PROGRAM AxisHorzMovementOutputCtrl_Arm1
VAR

	LdUnhook: CMP_OC_DW;
	Stn1Unhook: CMP_OC_DW;
	Stn2Unhook: CMP_OC_DW;
	Stn3Unhook: CMP_OC_DW;
	Stn4Unhook: CMP_OC_DW;
	Stn5Unhook: CMP_OC_DW;
	Stn6Unhook: CMP_OC_DW;
	Stn7Unhook: CMP_OC_DW;
	Stn8Unhook: CMP_OC_DW;
	Stn9Unhook: CMP_OC_DW;
	Stn10Unhook: CMP_OC_DW;
	Stn11Unhook: CMP_OC_DW;
	Stn12Unhook: CMP_OC_DW;
	Uld1Unhook: CMP_OC_DW;
	Uld2Unhook: CMP_OC_DW;

	LdHook: CMP_OC_DW;
	Stn1Hook: CMP_OC_DW;
	Stn2Hook: CMP_OC_DW;
	Stn3Hook: CMP_OC_DW;
	Stn4Hook: CMP_OC_DW;
	Stn5Hook: CMP_OC_DW;
	Stn6Hook: CMP_OC_DW;
	Stn7Hook: CMP_OC_DW;
	Stn8Hook: CMP_OC_DW;
	Stn9Hook: CMP_OC_DW;
	Stn10Hook: CMP_OC_DW;
	Stn11Hook: CMP_OC_DW;
	Stn12Hook: CMP_OC_DW;
	Uld1Hook: CMP_OC_DW;
	Uld2Hook: CMP_OC_DW;

END_VAR

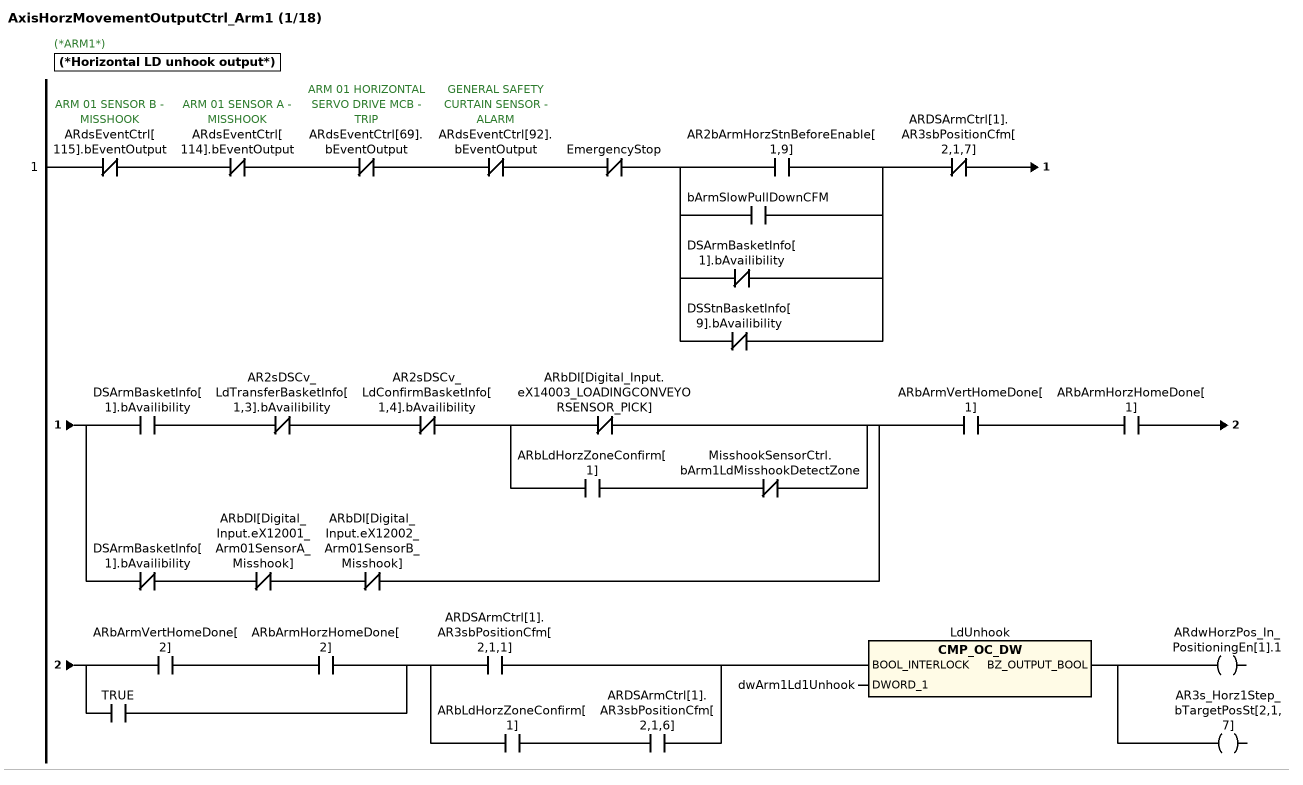
// NETWORK 1
// (*ARM1*)
//   ARdsEventCtrl[115].bEventOutput: ARM 01 SENSOR B - MISSHOOK
//   ARdsEventCtrl[114].bEventOutput: ARM 01 SENSOR A - MISSHOOK
//   ARdsEventCtrl[69].bEventOutput: ARM 01 HORIZONTAL SERVO DRIVE MCB - TRIP
//   ARdsEventCtrl[92].bEventOutput: GENERAL SAFETY CURTAIN SENSOR - ALARM
// label: (*Horizontal LD unhook output*)
LdUnhook(BOOL_INTERLOCK := (((NOT ARdsEventCtrl[115].bEventOutput AND NOT ARdsEventCtrl[114].bEventOutput AND NOT ARdsEventCtrl[69].bEventOutput AND NOT ARdsEventCtrl[92].bEventOutput AND NOT EmergencyStop) AND (AR2bArmHorzStnBeforeEnable[1,9] OR bArmSlowPullDownCFM OR NOT DSArmBasketInfo[1].bAvailibility OR NOT DSStnBasketInfo[9].bAvailibility)) AND NOT ARDSArmCtrl[1].AR3sbPositionCfm[2,1,7] AND (DSArmBasketInfo[1].bAvailibility AND NOT AR2sDSCv_LdTransferBasketInfo[1,3].bAvailibility AND NOT AR2sDSCv_LdConfirmBasketInfo[1,4].bAvailibility AND (NOT ARbDI[Digital_Input.eX14003_LOADINGCONVEYORSENSOR_PICK] OR ARbLdHorzZoneConfirm[1] AND NOT MisshookSensorCtrl.bArm1LdMisshookDetectZone) OR NOT DSArmBasketInfo[1].bAvailibility AND NOT ARbDI[Digital_Input.eX12001_Arm01SensorA_Misshook] AND NOT ARbDI[Digital_Input.eX12002_Arm01SensorB_Misshook])) AND ARbArmVertHomeDone[1] AND ARbArmHorzHomeDone[1] AND (ARbArmVertHomeDone[2] AND ARbArmHorzHomeDone[2] OR TRUE) AND (ARDSArmCtrl[1].AR3sbPositionCfm[2,1,1] OR ARbLdHorzZoneConfirm[1] AND ARDSArmCtrl[1].AR3sbPositionCfm[2,1,6]), DWORD_1 := dwArm1Ld1Unhook); // CMP_OC_DW
ARdwHorzPos_In_PositioningEn[1].1 := LdUnhook.BZ_OUTPUT_BOOL;
AR3s_Horz1Step_bTargetPosSt[2,1,7] := LdUnhook.BZ_OUTPUT_BOOL;

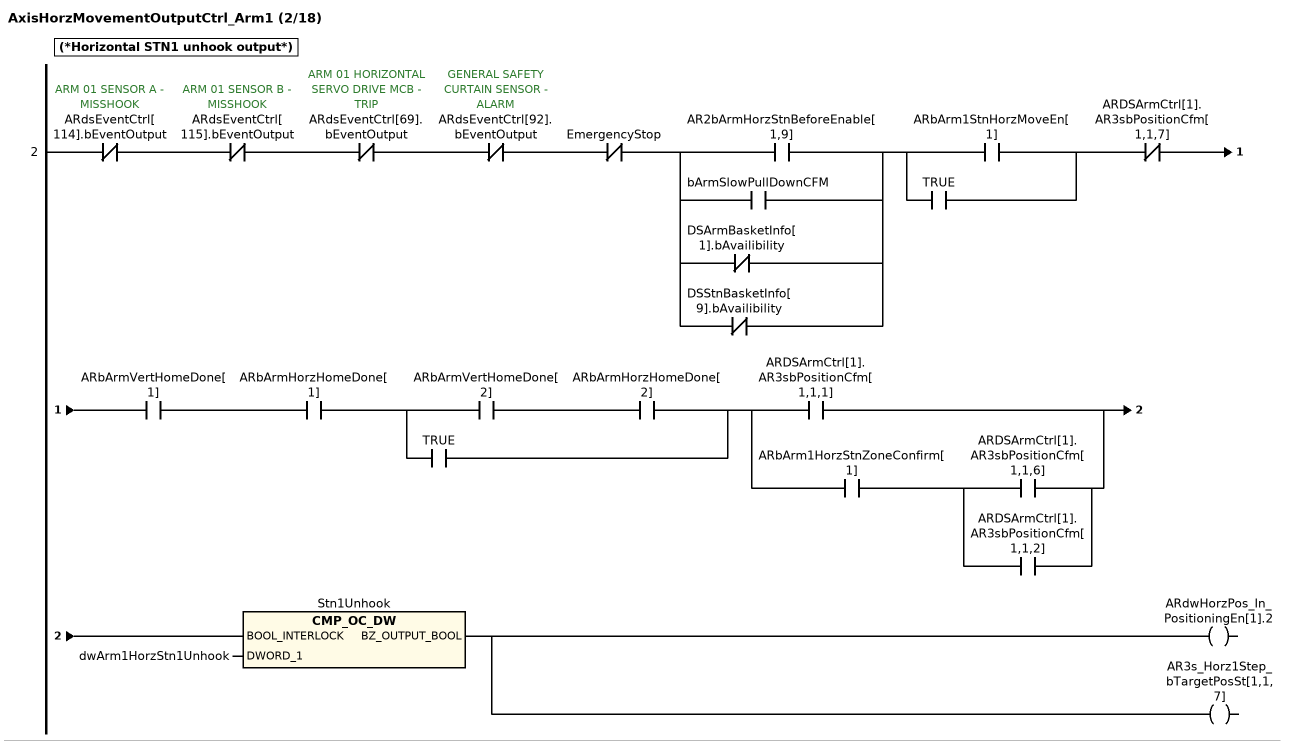
// NETWORK 2
//   ARdsEventCtrl[114].bEventOutput: ARM 01 SENSOR A - MISSHOOK
//   ARdsEventCtrl[115].bEventOutput: ARM 01 SENSOR B - MISSHOOK
//   ARdsEventCtrl[69].bEventOutput: ARM 01 HORIZONTAL SERVO DRIVE MCB - TRIP
//   ARdsEventCtrl[92].bEventOutput: GENERAL SAFETY CURTAIN SENSOR - ALARM
// label: (*Horizontal STN1 unhook output*)
Stn1Unhook(BOOL_INTERLOCK := ((NOT ARdsEventCtrl[114].bEventOutput AND NOT ARdsEventCtrl[115].bEventOutput AND NOT ARdsEventCtrl[69].bEventOutput AND NOT ARdsEventCtrl[92].bEventOutput AND NOT EmergencyStop) AND (AR2bArmHorzStnBeforeEnable[1,9] OR bArmSlowPullDownCFM OR NOT DSArmBasketInfo[1].bAvailibility OR NOT DSStnBasketInfo[9].bAvailibility) AND (ARbArm1StnHorzMoveEn[1] OR TRUE)) AND NOT ARDSArmCtrl[1].AR3sbPositionCfm[1,1,7] AND ARbArmVertHomeDone[1] AND ARbArmHorzHomeDone[1] AND (ARbArmVertHomeDone[2] AND ARbArmHorzHomeDone[2] OR TRUE) AND (ARDSArmCtrl[1].AR3sbPositionCfm[1,1,1] OR ARbArm1HorzStnZoneConfirm[1] AND (ARDSArmCtrl[1].AR3sbPositionCfm[1,1,6] OR ARDSArmCtrl[1].AR3sbPositionCfm[1,1,2])), DWORD_1 := dwArm1HorzStn1Unhook); // CMP_OC_DW
ARdwHorzPos_In_PositioningEn[1].2 := Stn1Unhook.BZ_OUTPUT_BOOL;
AR3s_Horz1Step_bTargetPosSt[1,1,7] := Stn1Unhook.BZ_OUTPUT_BOOL;

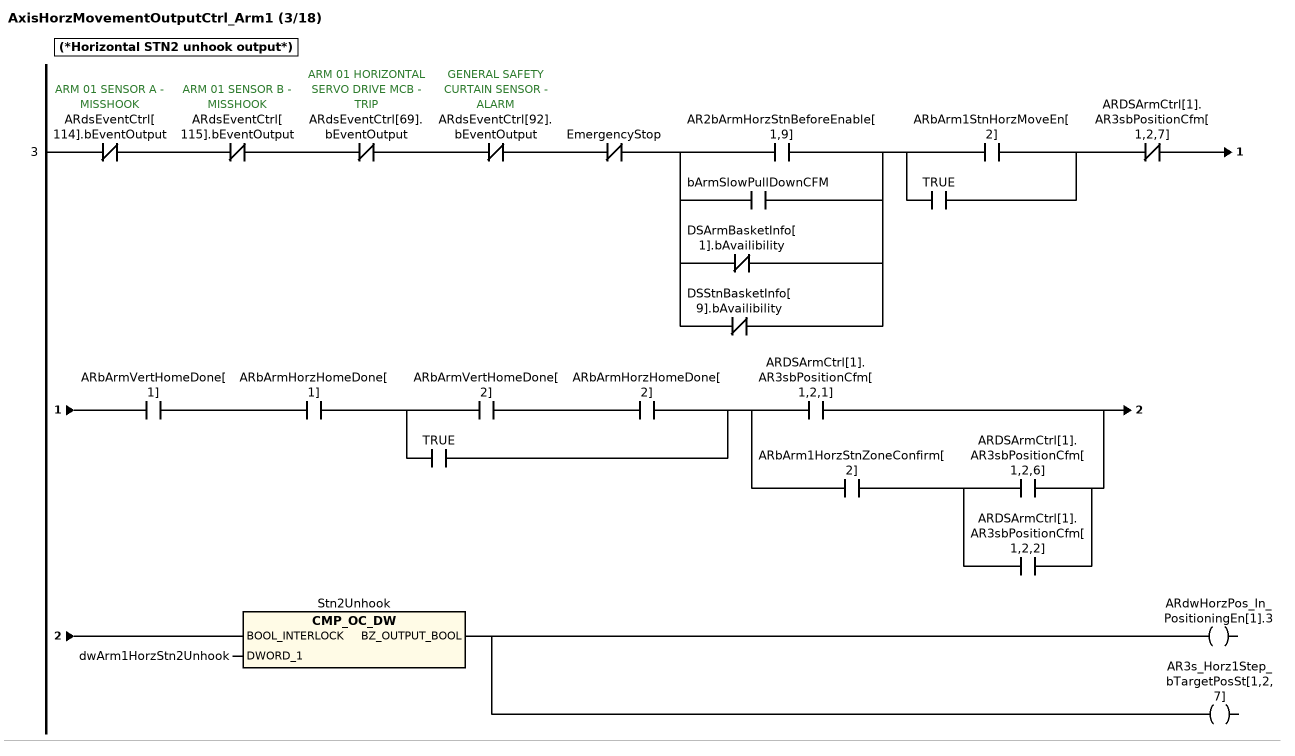
// NETWORK 3
//   ARdsEventCtrl[114].bEventOutput: ARM 01 SENSOR A - MISSHOOK
//   ARdsEventCtrl[115].bEventOutput: ARM 01 SENSOR B - MISSHOOK
//   ARdsEventCtrl[69].bEventOutput: ARM 01 HORIZONTAL SERVO DRIVE MCB - TRIP
//   ARdsEventCtrl[92].bEventOutput: GENERAL SAFETY CURTAIN SENSOR - ALARM
// label: (*Horizontal STN2 unhook output*)
Stn2Unhook(BOOL_INTERLOCK := ((NOT ARdsEventCtrl[114].bEventOutput AND NOT ARdsEventCtrl[115].bEventOutput AND NOT ARdsEventCtrl[69].bEventOutput AND NOT ARdsEventCtrl[92].bEventOutput AND NOT EmergencyStop) AND (AR2bArmHorzStnBeforeEnable[1,9] OR bArmSlowPullDownCFM OR NOT DSArmBasketInfo[1].bAvailibility OR NOT DSStnBasketInfo[9].bAvailibility) AND (ARbArm1StnHorzMoveEn[2] OR TRUE)) AND NOT ARDSArmCtrl[1].AR3sbPositionCfm[1,2,7] AND ARbArmVertHomeDone[1] AND ARbArmHorzHomeDone[1] AND (ARbArmVertHomeDone[2] AND ARbArmHorzHomeDone[2] OR TRUE) AND (ARDSArmCtrl[1].AR3sbPositionCfm[1,2,1] OR ARbArm1HorzStnZoneConfirm[2] AND (ARDSArmCtrl[1].AR3sbPositionCfm[1,2,6] OR ARDSArmCtrl[1].AR3sbPositionCfm[1,2,2])), DWORD_1 := dwArm1HorzStn2Unhook); // CMP_OC_DW
ARdwHorzPos_In_PositioningEn[1].3 := Stn2Unhook.BZ_OUTPUT_BOOL;
AR3s_Horz1Step_bTargetPosSt[1,2,7] := Stn2Unhook.BZ_OUTPUT_BOOL;

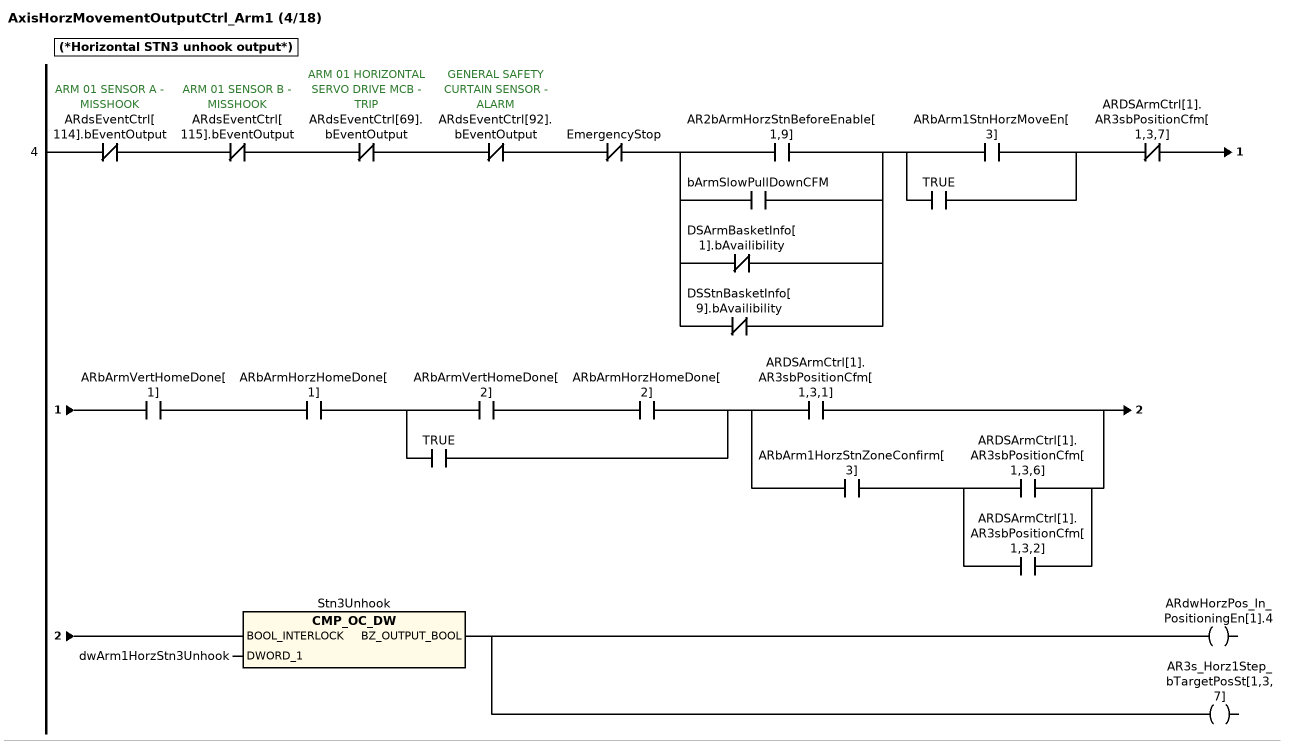
// NETWORK 4
//   ARdsEventCtrl[114].bEventOutput: ARM 01 SENSOR A - MISSHOOK
//   ARdsEventCtrl[115].bEventOutput: ARM 01 SENSOR B - MISSHOOK
//   ARdsEventCtrl[69].bEventOutput: ARM 01 HORIZONTAL SERVO DRIVE MCB - TRIP
//   ARdsEventCtrl[92].bEventOutput: GENERAL SAFETY CURTAIN SENSOR - ALARM
// label: (*Horizontal STN3 unhook output*)
Stn3Unhook(BOOL_INTERLOCK := ((NOT ARdsEventCtrl[114].bEventOutput AND NOT ARdsEventCtrl[115].bEventOutput AND NOT ARdsEventCtrl[69].bEventOutput AND NOT ARdsEventCtrl[92].bEventOutput AND NOT EmergencyStop) AND (AR2bArmHorzStnBeforeEnable[1,9] OR bArmSlowPullDownCFM OR NOT DSArmBasketInfo[1].bAvailibility OR NOT DSStnBasketInfo[9].bAvailibility) AND (ARbArm1StnHorzMoveEn[3] OR TRUE)) AND NOT ARDSArmCtrl[1].AR3sbPositionCfm[1,3,7] AND ARbArmVertHomeDone[1] AND ARbArmHorzHomeDone[1] AND (ARbArmVertHomeDone[2] AND ARbArmHorzHomeDone[2] OR TRUE) AND (ARDSArmCtrl[1].AR3sbPositionCfm[1,3,1] OR ARbArm1HorzStnZoneConfirm[3] AND (ARDSArmCtrl[1].AR3sbPositionCfm[1,3,6] OR ARDSArmCtrl[1].AR3sbPositionCfm[1,3,2])), DWORD_1 := dwArm1HorzStn3Unhook); // CMP_OC_DW
ARdwHorzPos_In_PositioningEn[1].4 := Stn3Unhook.BZ_OUTPUT_BOOL;
AR3s_Horz1Step_bTargetPosSt[1,3,7] := Stn3Unhook.BZ_OUTPUT_BOOL;

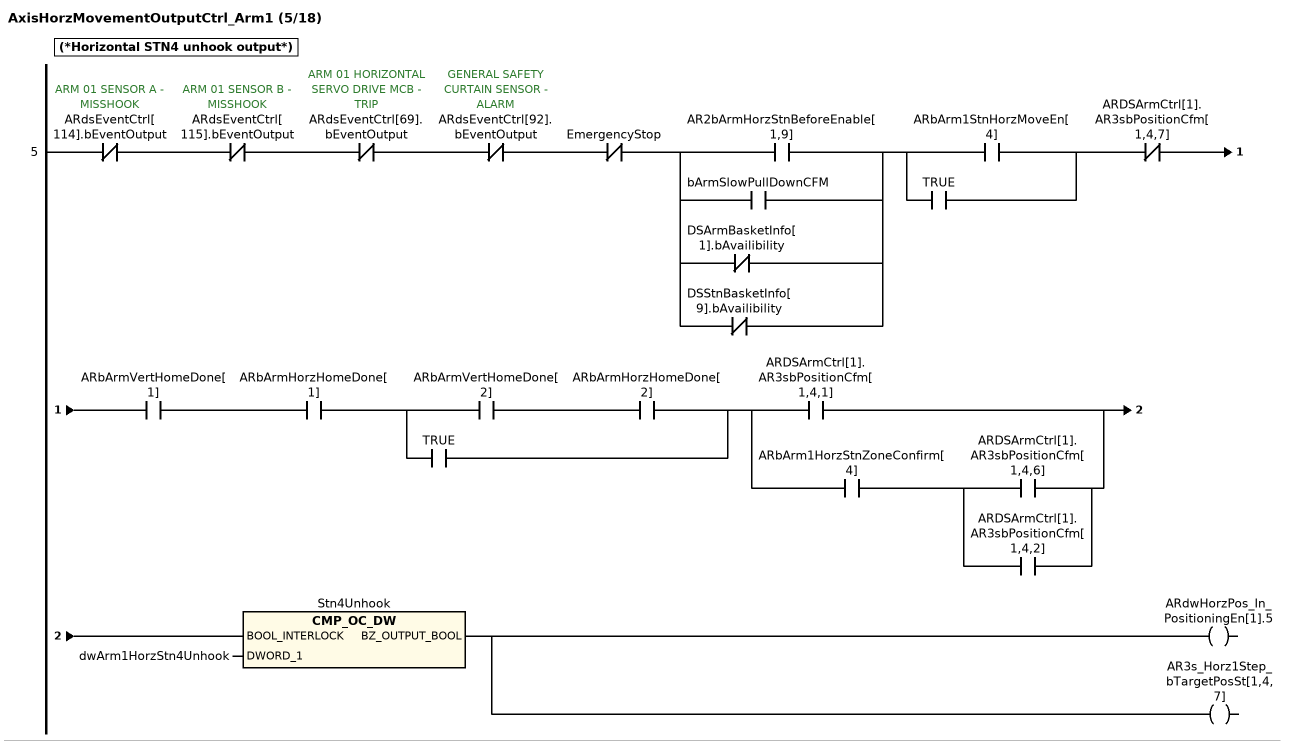
// NETWORK 5
//   ARdsEventCtrl[114].bEventOutput: ARM 01 SENSOR A - MISSHOOK
//   ARdsEventCtrl[115].bEventOutput: ARM 01 SENSOR B - MISSHOOK
//   ARdsEventCtrl[69].bEventOutput: ARM 01 HORIZONTAL SERVO DRIVE MCB - TRIP
//   ARdsEventCtrl[92].bEventOutput: GENERAL SAFETY CURTAIN SENSOR - ALARM
// label: (*Horizontal STN4 unhook output*)
Stn4Unhook(BOOL_INTERLOCK := ((NOT ARdsEventCtrl[114].bEventOutput AND NOT ARdsEventCtrl[115].bEventOutput AND NOT ARdsEventCtrl[69].bEventOutput AND NOT ARdsEventCtrl[92].bEventOutput AND NOT EmergencyStop) AND (AR2bArmHorzStnBeforeEnable[1,9] OR bArmSlowPullDownCFM OR NOT DSArmBasketInfo[1].bAvailibility OR NOT DSStnBasketInfo[9].bAvailibility) AND (ARbArm1StnHorzMoveEn[4] OR TRUE)) AND NOT ARDSArmCtrl[1].AR3sbPositionCfm[1,4,7] AND ARbArmVertHomeDone[1] AND ARbArmHorzHomeDone[1] AND (ARbArmVertHomeDone[2] AND ARbArmHorzHomeDone[2] OR TRUE) AND (ARDSArmCtrl[1].AR3sbPositionCfm[1,4,1] OR ARbArm1HorzStnZoneConfirm[4] AND (ARDSArmCtrl[1].AR3sbPositionCfm[1,4,6] OR ARDSArmCtrl[1].AR3sbPositionCfm[1,4,2])), DWORD_1 := dwArm1HorzStn4Unhook); // CMP_OC_DW
ARdwHorzPos_In_PositioningEn[1].5 := Stn4Unhook.BZ_OUTPUT_BOOL;
AR3s_Horz1Step_bTargetPosSt[1,4,7] := Stn4Unhook.BZ_OUTPUT_BOOL;

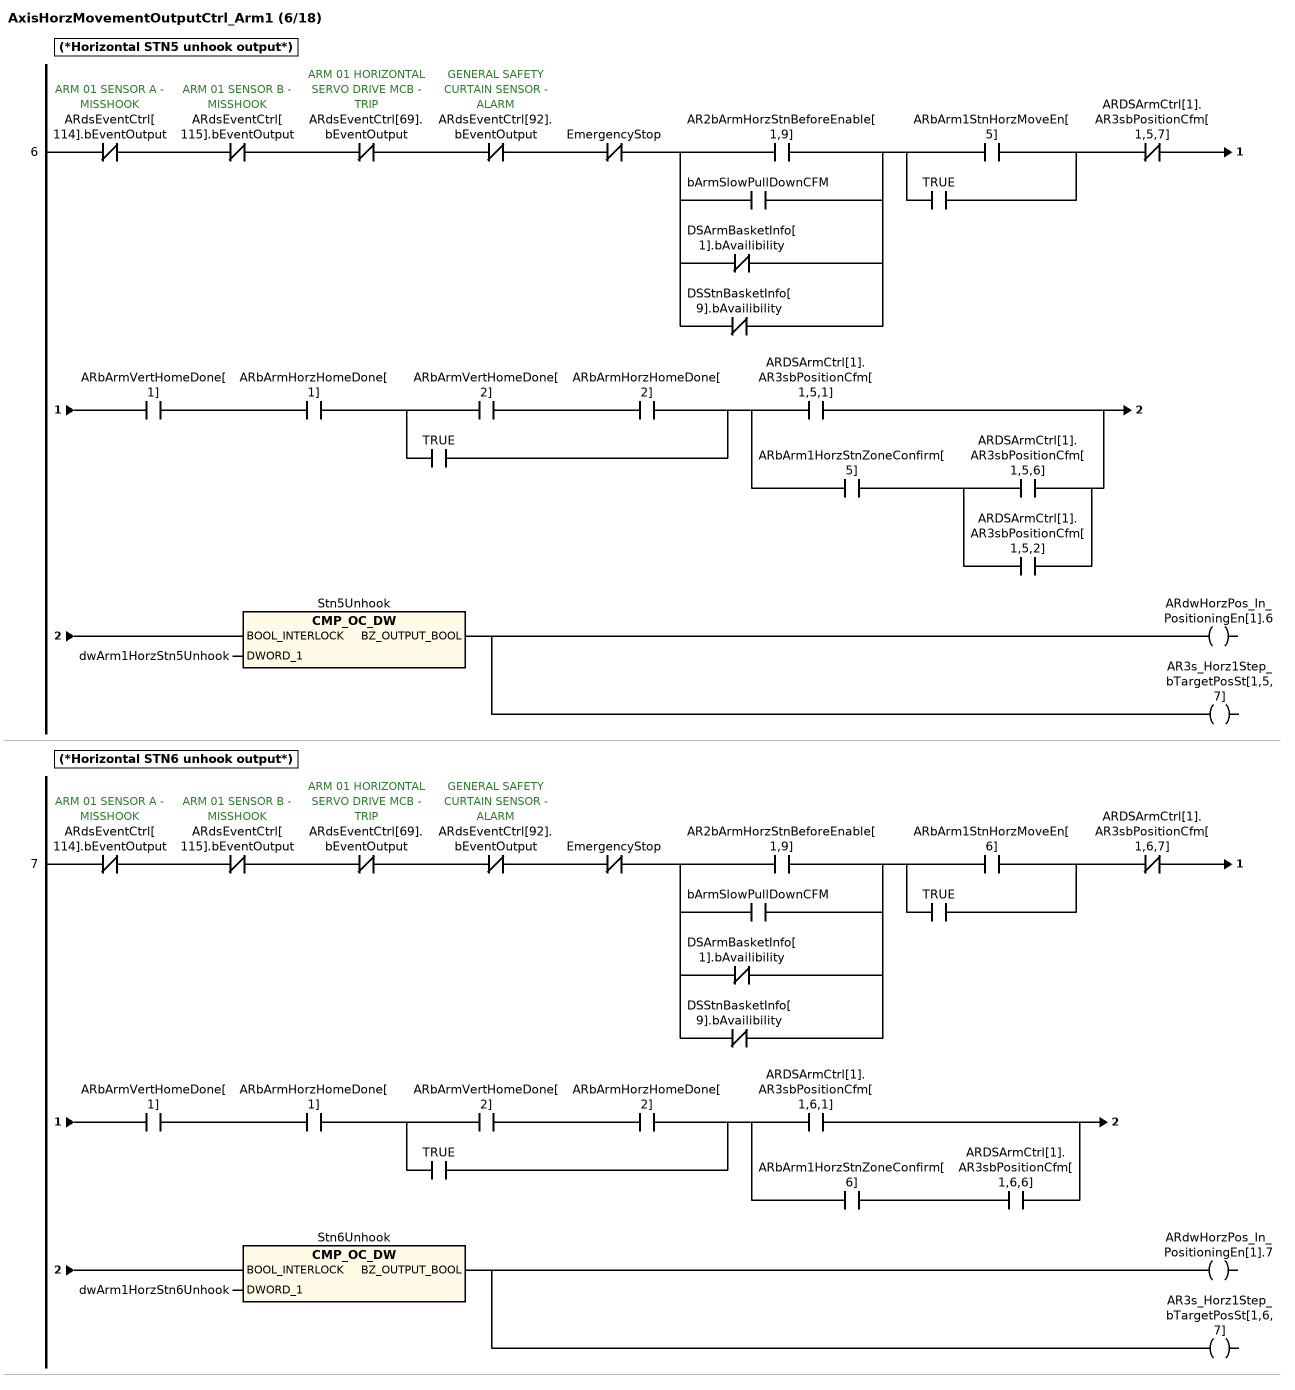
// NETWORK 6
//   ARdsEventCtrl[114].bEventOutput: ARM 01 SENSOR A - MISSHOOK
//   ARdsEventCtrl[115].bEventOutput: ARM 01 SENSOR B - MISSHOOK
//   ARdsEventCtrl[69].bEventOutput: ARM 01 HORIZONTAL SERVO DRIVE MCB - TRIP
//   ARdsEventCtrl[92].bEventOutput: GENERAL SAFETY CURTAIN SENSOR - ALARM
// label: (*Horizontal STN5 unhook output*)
Stn5Unhook(BOOL_INTERLOCK := ((NOT ARdsEventCtrl[114].bEventOutput AND NOT ARdsEventCtrl[115].bEventOutput AND NOT ARdsEventCtrl[69].bEventOutput AND NOT ARdsEventCtrl[92].bEventOutput AND NOT EmergencyStop) AND (AR2bArmHorzStnBeforeEnable[1,9] OR bArmSlowPullDownCFM OR NOT DSArmBasketInfo[1].bAvailibility OR NOT DSStnBasketInfo[9].bAvailibility) AND (ARbArm1StnHorzMoveEn[5] OR TRUE)) AND NOT ARDSArmCtrl[1].AR3sbPositionCfm[1,5,7] AND ARbArmVertHomeDone[1] AND ARbArmHorzHomeDone[1] AND (ARbArmVertHomeDone[2] AND ARbArmHorzHomeDone[2] OR TRUE) AND (ARDSArmCtrl[1].AR3sbPositionCfm[1,5,1] OR ARbArm1HorzStnZoneConfirm[5] AND (ARDSArmCtrl[1].AR3sbPositionCfm[1,5,6] OR ARDSArmCtrl[1].AR3sbPositionCfm[1,5,2])), DWORD_1 := dwArm1HorzStn5Unhook); // CMP_OC_DW
ARdwHorzPos_In_PositioningEn[1].6 := Stn5Unhook.BZ_OUTPUT_BOOL;
AR3s_Horz1Step_bTargetPosSt[1,5,7] := Stn5Unhook.BZ_OUTPUT_BOOL;

// NETWORK 7
//   ARdsEventCtrl[114].bEventOutput: ARM 01 SENSOR A - MISSHOOK
//   ARdsEventCtrl[115].bEventOutput: ARM 01 SENSOR B - MISSHOOK
//   ARdsEventCtrl[69].bEventOutput: ARM 01 HORIZONTAL SERVO DRIVE MCB - TRIP
//   ARdsEventCtrl[92].bEventOutput: GENERAL SAFETY CURTAIN SENSOR - ALARM
// label: (*Horizontal STN6 unhook output*)
Stn6Unhook(BOOL_INTERLOCK := ((NOT ARdsEventCtrl[114].bEventOutput AND NOT ARdsEventCtrl[115].bEventOutput AND NOT ARdsEventCtrl[69].bEventOutput AND NOT ARdsEventCtrl[92].bEventOutput AND NOT EmergencyStop) AND ((AR2bArmHorzStnBeforeEnable[1,9] OR bArmSlowPullDownCFM OR NOT DSArmBasketInfo[1].bAvailibility OR NOT DSStnBasketInfo[9].bAvailibility) AND (ARbArm1StnHorzMoveEn[6] OR TRUE))) AND NOT ARDSArmCtrl[1].AR3sbPositionCfm[1,6,7] AND ARbArmVertHomeDone[1] AND ARbArmHorzHomeDone[1] AND (ARbArmVertHomeDone[2] AND ARbArmHorzHomeDone[2] OR TRUE) AND (ARDSArmCtrl[1].AR3sbPositionCfm[1,6,1] OR ARbArm1HorzStnZoneConfirm[6] AND ARDSArmCtrl[1].AR3sbPositionCfm[1,6,6]), DWORD_1 := dwArm1HorzStn6Unhook); // CMP_OC_DW
ARdwHorzPos_In_PositioningEn[1].7 := Stn6Unhook.BZ_OUTPUT_BOOL;
AR3s_Horz1Step_bTargetPosSt[1,6,7] := Stn6Unhook.BZ_OUTPUT_BOOL;

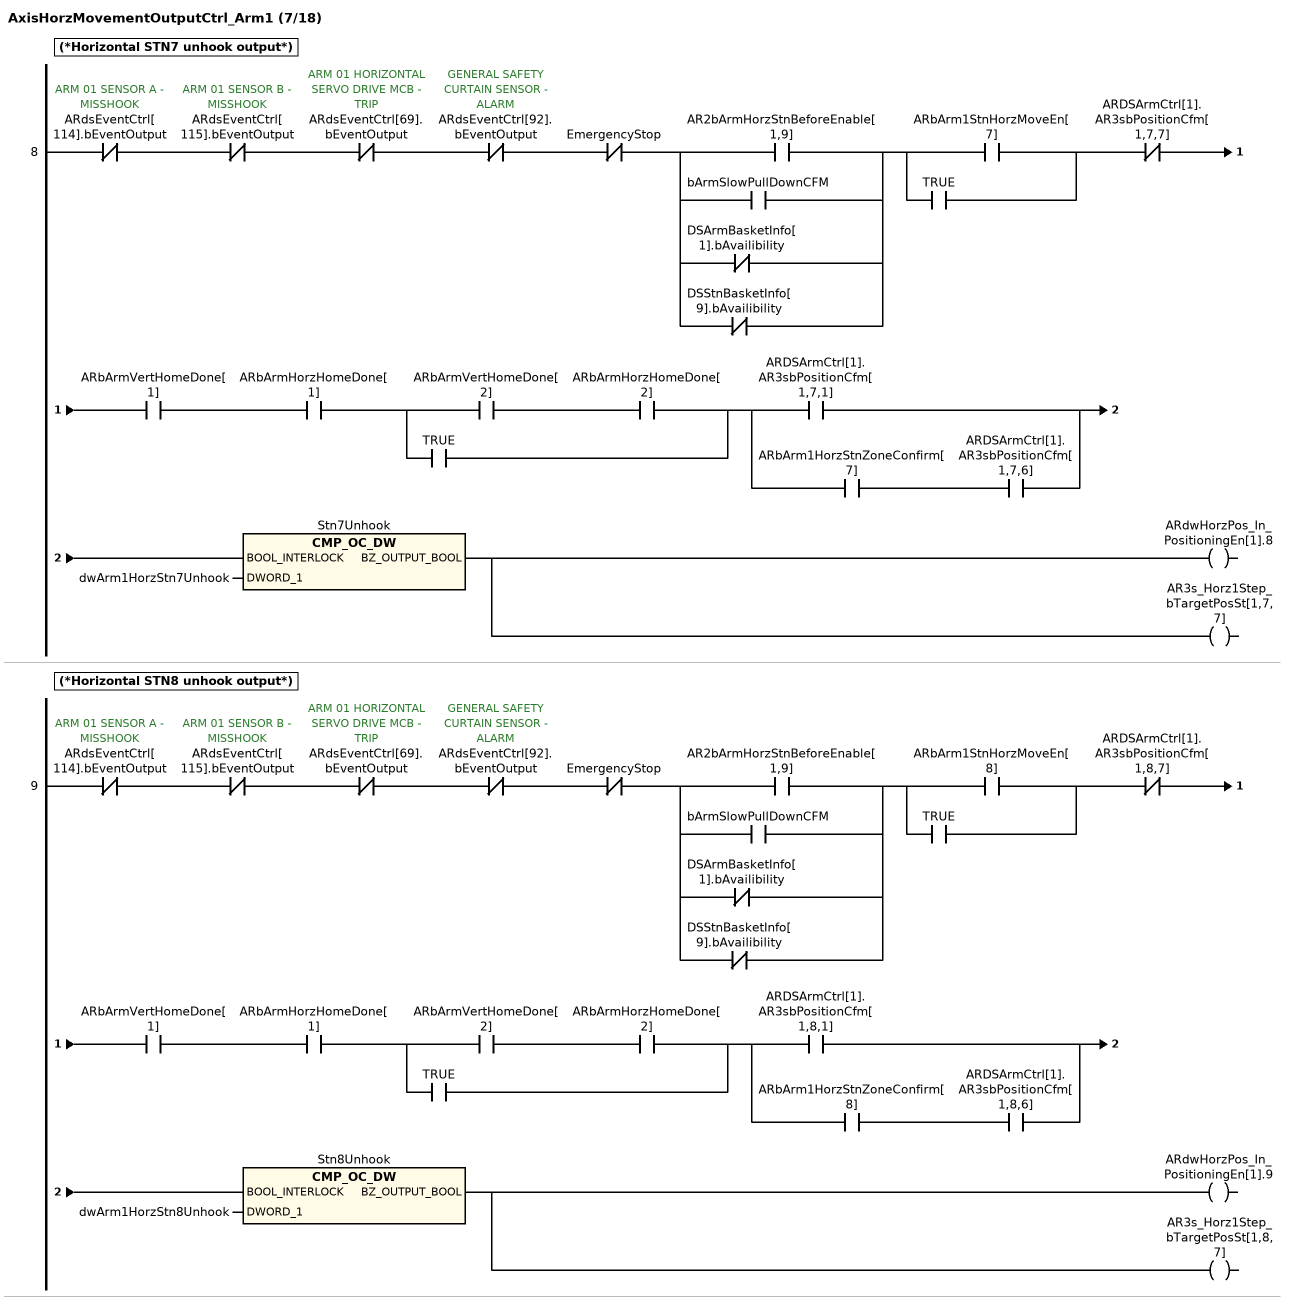
// NETWORK 8
//   ARdsEventCtrl[114].bEventOutput: ARM 01 SENSOR A - MISSHOOK
//   ARdsEventCtrl[115].bEventOutput: ARM 01 SENSOR B - MISSHOOK
//   ARdsEventCtrl[69].bEventOutput: ARM 01 HORIZONTAL SERVO DRIVE MCB - TRIP
//   ARdsEventCtrl[92].bEventOutput: GENERAL SAFETY CURTAIN SENSOR - ALARM
// label: (*Horizontal STN7 unhook output*)
Stn7Unhook(BOOL_INTERLOCK := ((NOT ARdsEventCtrl[114].bEventOutput AND NOT ARdsEventCtrl[115].bEventOutput AND NOT ARdsEventCtrl[69].bEventOutput AND NOT ARdsEventCtrl[92].bEventOutput AND NOT EmergencyStop) AND (AR2bArmHorzStnBeforeEnable[1,9] OR bArmSlowPullDownCFM OR NOT DSArmBasketInfo[1].bAvailibility OR NOT DSStnBasketInfo[9].bAvailibility) AND (ARbArm1StnHorzMoveEn[7] OR TRUE)) AND NOT ARDSArmCtrl[1].AR3sbPositionCfm[1,7,7] AND ARbArmVertHomeDone[1] AND ARbArmHorzHomeDone[1] AND (ARbArmVertHomeDone[2] AND ARbArmHorzHomeDone[2] OR TRUE) AND (ARDSArmCtrl[1].AR3sbPositionCfm[1,7,1] OR ARbArm1HorzStnZoneConfirm[7] AND ARDSArmCtrl[1].AR3sbPositionCfm[1,7,6]), DWORD_1 := dwArm1HorzStn7Unhook); // CMP_OC_DW
ARdwHorzPos_In_PositioningEn[1].8 := Stn7Unhook.BZ_OUTPUT_BOOL;
AR3s_Horz1Step_bTargetPosSt[1,7,7] := Stn7Unhook.BZ_OUTPUT_BOOL;

// NETWORK 9
//   ARdsEventCtrl[114].bEventOutput: ARM 01 SENSOR A - MISSHOOK
//   ARdsEventCtrl[115].bEventOutput: ARM 01 SENSOR B - MISSHOOK
//   ARdsEventCtrl[69].bEventOutput: ARM 01 HORIZONTAL SERVO DRIVE MCB - TRIP
//   ARdsEventCtrl[92].bEventOutput: GENERAL SAFETY CURTAIN SENSOR - ALARM
// label: (*Horizontal STN8 unhook output*)
Stn8Unhook(BOOL_INTERLOCK := ((NOT ARdsEventCtrl[114].bEventOutput AND NOT ARdsEventCtrl[115].bEventOutput AND NOT ARdsEventCtrl[69].bEventOutput AND NOT ARdsEventCtrl[92].bEventOutput AND NOT EmergencyStop) AND (AR2bArmHorzStnBeforeEnable[1,9] OR bArmSlowPullDownCFM OR NOT DSArmBasketInfo[1].bAvailibility OR NOT DSStnBasketInfo[9].bAvailibility) AND (ARbArm1StnHorzMoveEn[8] OR TRUE)) AND NOT ARDSArmCtrl[1].AR3sbPositionCfm[1,8,7] AND ARbArmVertHomeDone[1] AND ARbArmHorzHomeDone[1] AND (ARbArmVertHomeDone[2] AND ARbArmHorzHomeDone[2] OR TRUE) AND (ARDSArmCtrl[1].AR3sbPositionCfm[1,8,1] OR ARbArm1HorzStnZoneConfirm[8] AND ARDSArmCtrl[1].AR3sbPositionCfm[1,8,6]), DWORD_1 := dwArm1HorzStn8Unhook); // CMP_OC_DW
ARdwHorzPos_In_PositioningEn[1].9 := Stn8Unhook.BZ_OUTPUT_BOOL;
AR3s_Horz1Step_bTargetPosSt[1,8,7] := Stn8Unhook.BZ_OUTPUT_BOOL;

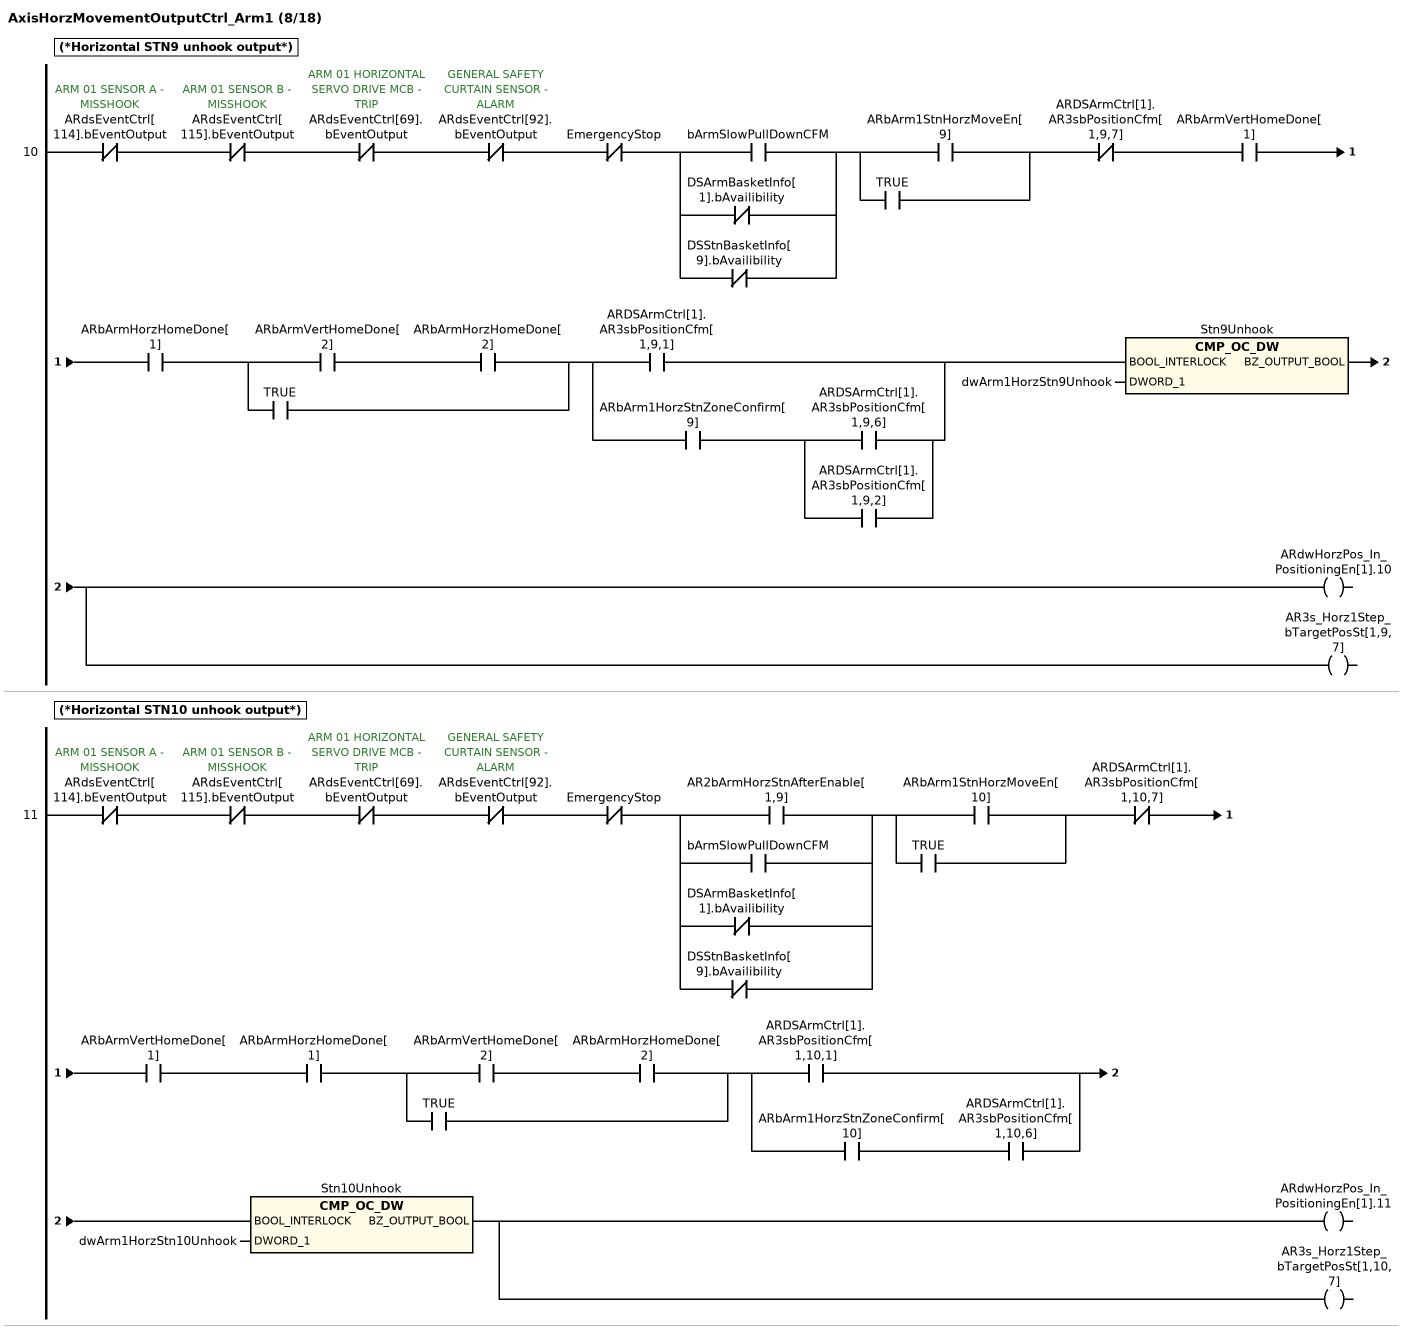
// NETWORK 10
//   ARdsEventCtrl[114].bEventOutput: ARM 01 SENSOR A - MISSHOOK
//   ARdsEventCtrl[115].bEventOutput: ARM 01 SENSOR B - MISSHOOK
//   ARdsEventCtrl[69].bEventOutput: ARM 01 HORIZONTAL SERVO DRIVE MCB - TRIP
//   ARdsEventCtrl[92].bEventOutput: GENERAL SAFETY CURTAIN SENSOR - ALARM
// label: (*Horizontal STN9 unhook output*)
Stn9Unhook(BOOL_INTERLOCK := ((NOT ARdsEventCtrl[114].bEventOutput AND NOT ARdsEventCtrl[115].bEventOutput AND NOT ARdsEventCtrl[69].bEventOutput AND NOT ARdsEventCtrl[92].bEventOutput AND NOT EmergencyStop) AND (bArmSlowPullDownCFM OR NOT DSArmBasketInfo[1].bAvailibility OR NOT DSStnBasketInfo[9].bAvailibility) AND (ARbArm1StnHorzMoveEn[9] OR TRUE)) AND NOT ARDSArmCtrl[1].AR3sbPositionCfm[1,9,7] AND ARbArmVertHomeDone[1] AND ARbArmHorzHomeDone[1] AND (ARbArmVertHomeDone[2] AND ARbArmHorzHomeDone[2] OR TRUE) AND (ARDSArmCtrl[1].AR3sbPositionCfm[1,9,1] OR ARbArm1HorzStnZoneConfirm[9] AND (ARDSArmCtrl[1].AR3sbPositionCfm[1,9,6] OR ARDSArmCtrl[1].AR3sbPositionCfm[1,9,2])), DWORD_1 := dwArm1HorzStn9Unhook); // CMP_OC_DW
ARdwHorzPos_In_PositioningEn[1].10 := Stn9Unhook.BZ_OUTPUT_BOOL;
AR3s_Horz1Step_bTargetPosSt[1,9,7] := Stn9Unhook.BZ_OUTPUT_BOOL;

// NETWORK 11
//   ARdsEventCtrl[114].bEventOutput: ARM 01 SENSOR A - MISSHOOK
//   ARdsEventCtrl[115].bEventOutput: ARM 01 SENSOR B - MISSHOOK
//   ARdsEventCtrl[69].bEventOutput: ARM 01 HORIZONTAL SERVO DRIVE MCB - TRIP
//   ARdsEventCtrl[92].bEventOutput: GENERAL SAFETY CURTAIN SENSOR - ALARM
// label: (*Horizontal STN10 unhook output*)
Stn10Unhook(BOOL_INTERLOCK := ((NOT ARdsEventCtrl[114].bEventOutput AND NOT ARdsEventCtrl[115].bEventOutput AND NOT ARdsEventCtrl[69].bEventOutput AND NOT ARdsEventCtrl[92].bEventOutput AND NOT EmergencyStop) AND (AR2bArmHorzStnAfterEnable[1,9] OR bArmSlowPullDownCFM OR NOT DSArmBasketInfo[1].bAvailibility OR NOT DSStnBasketInfo[9].bAvailibility) AND (ARbArm1StnHorzMoveEn[10] OR TRUE)) AND NOT ARDSArmCtrl[1].AR3sbPositionCfm[1,10,7] AND ARbArmVertHomeDone[1] AND ARbArmHorzHomeDone[1] AND (ARbArmVertHomeDone[2] AND ARbArmHorzHomeDone[2] OR TRUE) AND (ARDSArmCtrl[1].AR3sbPositionCfm[1,10,1] OR ARbArm1HorzStnZoneConfirm[10] AND ARDSArmCtrl[1].AR3sbPositionCfm[1,10,6]), DWORD_1 := dwArm1HorzStn10Unhook); // CMP_OC_DW
ARdwHorzPos_In_PositioningEn[1].11 := Stn10Unhook.BZ_OUTPUT_BOOL;
AR3s_Horz1Step_bTargetPosSt[1,10,7] := Stn10Unhook.BZ_OUTPUT_BOOL;

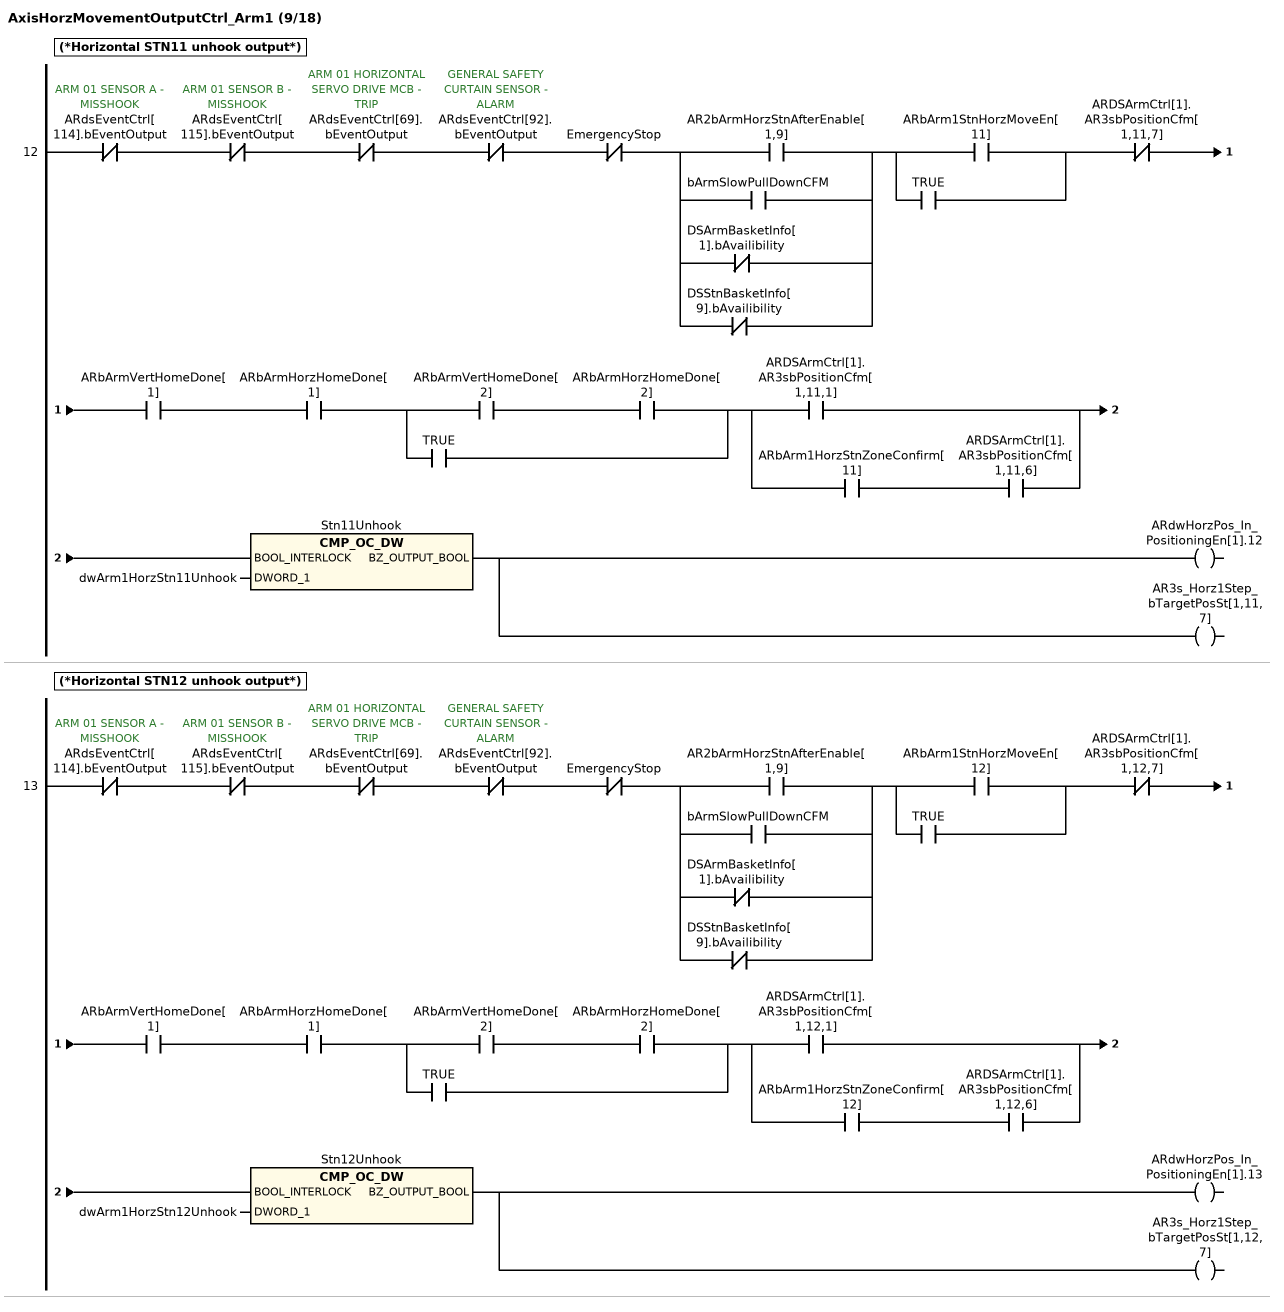
// NETWORK 12
//   ARdsEventCtrl[114].bEventOutput: ARM 01 SENSOR A - MISSHOOK
//   ARdsEventCtrl[115].bEventOutput: ARM 01 SENSOR B - MISSHOOK
//   ARdsEventCtrl[69].bEventOutput: ARM 01 HORIZONTAL SERVO DRIVE MCB - TRIP
//   ARdsEventCtrl[92].bEventOutput: GENERAL SAFETY CURTAIN SENSOR - ALARM
// label: (*Horizontal STN11 unhook output*)
Stn11Unhook(BOOL_INTERLOCK := ((NOT ARdsEventCtrl[114].bEventOutput AND NOT ARdsEventCtrl[115].bEventOutput AND NOT ARdsEventCtrl[69].bEventOutput AND NOT ARdsEventCtrl[92].bEventOutput AND NOT EmergencyStop) AND (AR2bArmHorzStnAfterEnable[1,9] OR bArmSlowPullDownCFM OR NOT DSArmBasketInfo[1].bAvailibility OR NOT DSStnBasketInfo[9].bAvailibility) AND (ARbArm1StnHorzMoveEn[11] OR TRUE)) AND NOT ARDSArmCtrl[1].AR3sbPositionCfm[1,11,7] AND ARbArmVertHomeDone[1] AND ARbArmHorzHomeDone[1] AND (ARbArmVertHomeDone[2] AND ARbArmHorzHomeDone[2] OR TRUE) AND (ARDSArmCtrl[1].AR3sbPositionCfm[1,11,1] OR ARbArm1HorzStnZoneConfirm[11] AND ARDSArmCtrl[1].AR3sbPositionCfm[1,11,6]), DWORD_1 := dwArm1HorzStn11Unhook); // CMP_OC_DW
ARdwHorzPos_In_PositioningEn[1].12 := Stn11Unhook.BZ_OUTPUT_BOOL;
AR3s_Horz1Step_bTargetPosSt[1,11,7] := Stn11Unhook.BZ_OUTPUT_BOOL;

// NETWORK 13
//   ARdsEventCtrl[114].bEventOutput: ARM 01 SENSOR A - MISSHOOK
//   ARdsEventCtrl[115].bEventOutput: ARM 01 SENSOR B - MISSHOOK
//   ARdsEventCtrl[69].bEventOutput: ARM 01 HORIZONTAL SERVO DRIVE MCB - TRIP
//   ARdsEventCtrl[92].bEventOutput: GENERAL SAFETY CURTAIN SENSOR - ALARM
// label: (*Horizontal STN12 unhook output*)
Stn12Unhook(BOOL_INTERLOCK := ((NOT ARdsEventCtrl[114].bEventOutput AND NOT ARdsEventCtrl[115].bEventOutput AND NOT ARdsEventCtrl[69].bEventOutput AND NOT ARdsEventCtrl[92].bEventOutput AND NOT EmergencyStop) AND (AR2bArmHorzStnAfterEnable[1,9] OR bArmSlowPullDownCFM OR NOT DSArmBasketInfo[1].bAvailibility OR NOT DSStnBasketInfo[9].bAvailibility) AND (ARbArm1StnHorzMoveEn[12] OR TRUE)) AND NOT ARDSArmCtrl[1].AR3sbPositionCfm[1,12,7] AND ARbArmVertHomeDone[1] AND ARbArmHorzHomeDone[1] AND (ARbArmVertHomeDone[2] AND ARbArmHorzHomeDone[2] OR TRUE) AND (ARDSArmCtrl[1].AR3sbPositionCfm[1,12,1] OR ARbArm1HorzStnZoneConfirm[12] AND ARDSArmCtrl[1].AR3sbPositionCfm[1,12,6]), DWORD_1 := dwArm1HorzStn12Unhook); // CMP_OC_DW
ARdwHorzPos_In_PositioningEn[1].13 := Stn12Unhook.BZ_OUTPUT_BOOL;
AR3s_Horz1Step_bTargetPosSt[1,12,7] := Stn12Unhook.BZ_OUTPUT_BOOL;

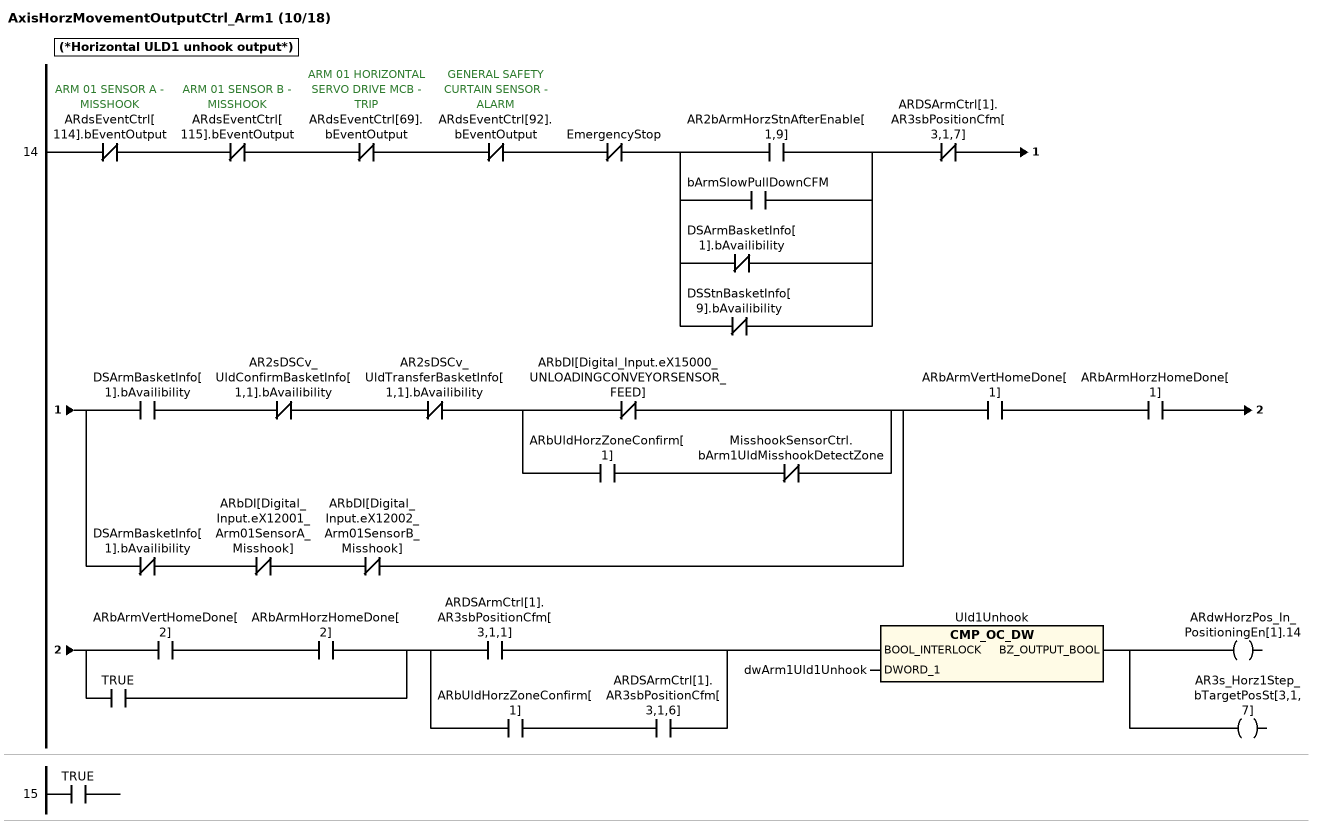
// NETWORK 14
//   ARdsEventCtrl[114].bEventOutput: ARM 01 SENSOR A - MISSHOOK
//   ARdsEventCtrl[115].bEventOutput: ARM 01 SENSOR B - MISSHOOK
//   ARdsEventCtrl[69].bEventOutput: ARM 01 HORIZONTAL SERVO DRIVE MCB - TRIP
//   ARdsEventCtrl[92].bEventOutput: GENERAL SAFETY CURTAIN SENSOR - ALARM
// label: (*Horizontal ULD1 unhook output*)
Uld1Unhook(BOOL_INTERLOCK := (((NOT ARdsEventCtrl[114].bEventOutput AND NOT ARdsEventCtrl[115].bEventOutput AND NOT ARdsEventCtrl[69].bEventOutput AND NOT ARdsEventCtrl[92].bEventOutput AND NOT EmergencyStop) AND (AR2bArmHorzStnAfterEnable[1,9] OR bArmSlowPullDownCFM OR NOT DSArmBasketInfo[1].bAvailibility OR NOT DSStnBasketInfo[9].bAvailibility)) AND NOT ARDSArmCtrl[1].AR3sbPositionCfm[3,1,7] AND (DSArmBasketInfo[1].bAvailibility AND NOT AR2sDSCv_UldConfirmBasketInfo[1,1].bAvailibility AND NOT AR2sDSCv_UldTransferBasketInfo[1,1].bAvailibility AND (NOT ARbDI[Digital_Input.eX15000_UNLOADINGCONVEYORSENSOR_FEED] OR ARbUldHorzZoneConfirm[1] AND NOT MisshookSensorCtrl.bArm1UldMisshookDetectZone) OR NOT DSArmBasketInfo[1].bAvailibility AND NOT ARbDI[Digital_Input.eX12001_Arm01SensorA_Misshook] AND NOT ARbDI[Digital_Input.eX12002_Arm01SensorB_Misshook])) AND ARbArmVertHomeDone[1] AND ARbArmHorzHomeDone[1] AND (ARbArmVertHomeDone[2] AND ARbArmHorzHomeDone[2] OR TRUE) AND (ARDSArmCtrl[1].AR3sbPositionCfm[3,1,1] OR ARbUldHorzZoneConfirm[1] AND ARDSArmCtrl[1].AR3sbPositionCfm[3,1,6]), DWORD_1 := dwArm1Uld1Unhook); // CMP_OC_DW
ARdwHorzPos_In_PositioningEn[1].14 := Uld1Unhook.BZ_OUTPUT_BOOL;
AR3s_Horz1Step_bTargetPosSt[3,1,7] := Uld1Unhook.BZ_OUTPUT_BOOL;

// NETWORK 15

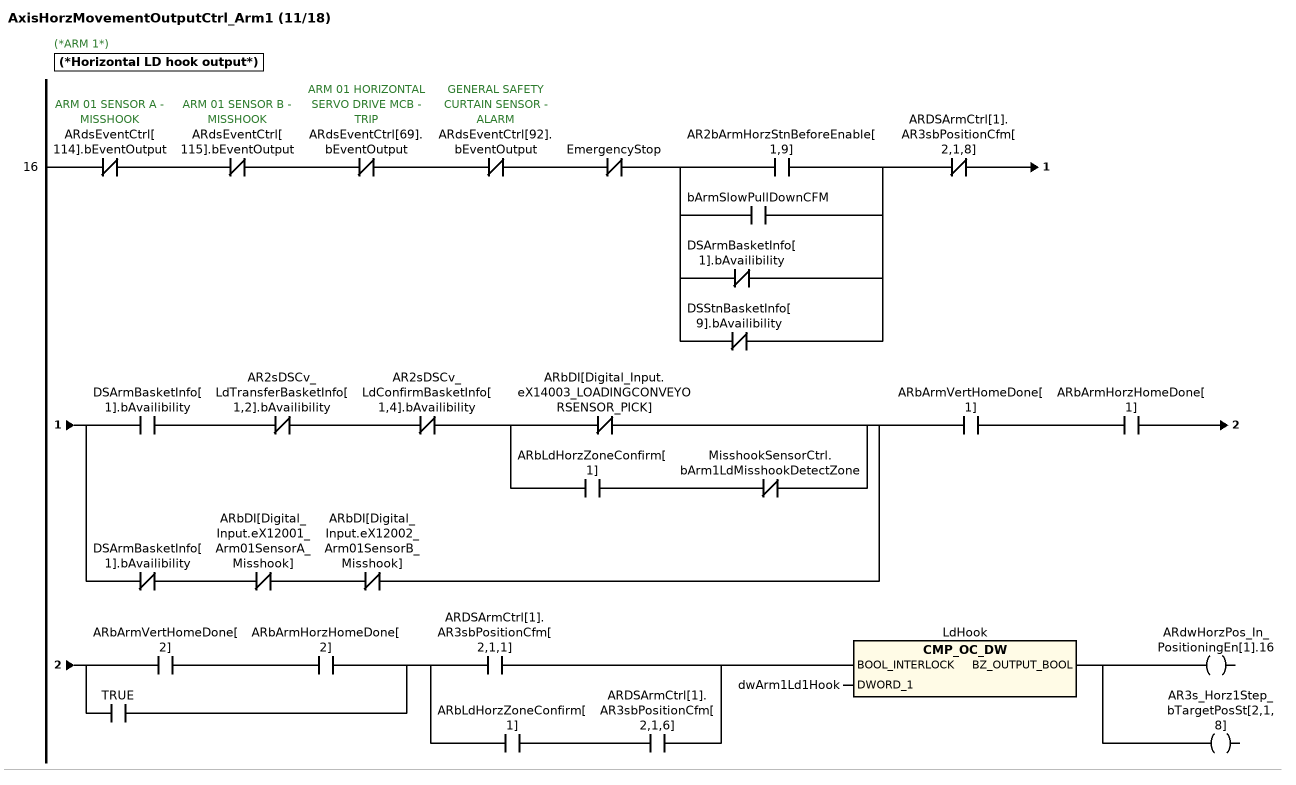
// NETWORK 16
// (*ARM 1*)
//   ARdsEventCtrl[114].bEventOutput: ARM 01 SENSOR A - MISSHOOK
//   ARdsEventCtrl[115].bEventOutput: ARM 01 SENSOR B - MISSHOOK
//   ARdsEventCtrl[69].bEventOutput: ARM 01 HORIZONTAL SERVO DRIVE MCB - TRIP
//   ARdsEventCtrl[92].bEventOutput: GENERAL SAFETY CURTAIN SENSOR - ALARM
// label: (*Horizontal LD hook output*)
LdHook(BOOL_INTERLOCK := (((NOT ARdsEventCtrl[114].bEventOutput AND NOT ARdsEventCtrl[115].bEventOutput AND NOT ARdsEventCtrl[69].bEventOutput AND NOT ARdsEventCtrl[92].bEventOutput AND NOT EmergencyStop) AND (AR2bArmHorzStnBeforeEnable[1,9] OR bArmSlowPullDownCFM OR NOT DSArmBasketInfo[1].bAvailibility OR NOT DSStnBasketInfo[9].bAvailibility)) AND NOT ARDSArmCtrl[1].AR3sbPositionCfm[2,1,8] AND (DSArmBasketInfo[1].bAvailibility AND NOT AR2sDSCv_LdTransferBasketInfo[1,2].bAvailibility AND NOT AR2sDSCv_LdConfirmBasketInfo[1,4].bAvailibility AND (NOT ARbDI[Digital_Input.eX14003_LOADINGCONVEYORSENSOR_PICK] OR ARbLdHorzZoneConfirm[1] AND NOT MisshookSensorCtrl.bArm1LdMisshookDetectZone) OR NOT DSArmBasketInfo[1].bAvailibility AND NOT ARbDI[Digital_Input.eX12001_Arm01SensorA_Misshook] AND NOT ARbDI[Digital_Input.eX12002_Arm01SensorB_Misshook])) AND ARbArmVertHomeDone[1] AND ARbArmHorzHomeDone[1] AND (ARbArmVertHomeDone[2] AND ARbArmHorzHomeDone[2] OR TRUE) AND (ARDSArmCtrl[1].AR3sbPositionCfm[2,1,1] OR ARbLdHorzZoneConfirm[1] AND ARDSArmCtrl[1].AR3sbPositionCfm[2,1,6]), DWORD_1 := dwArm1Ld1Hook); // CMP_OC_DW
ARdwHorzPos_In_PositioningEn[1].16 := LdHook.BZ_OUTPUT_BOOL;
AR3s_Horz1Step_bTargetPosSt[2,1,8] := LdHook.BZ_OUTPUT_BOOL;

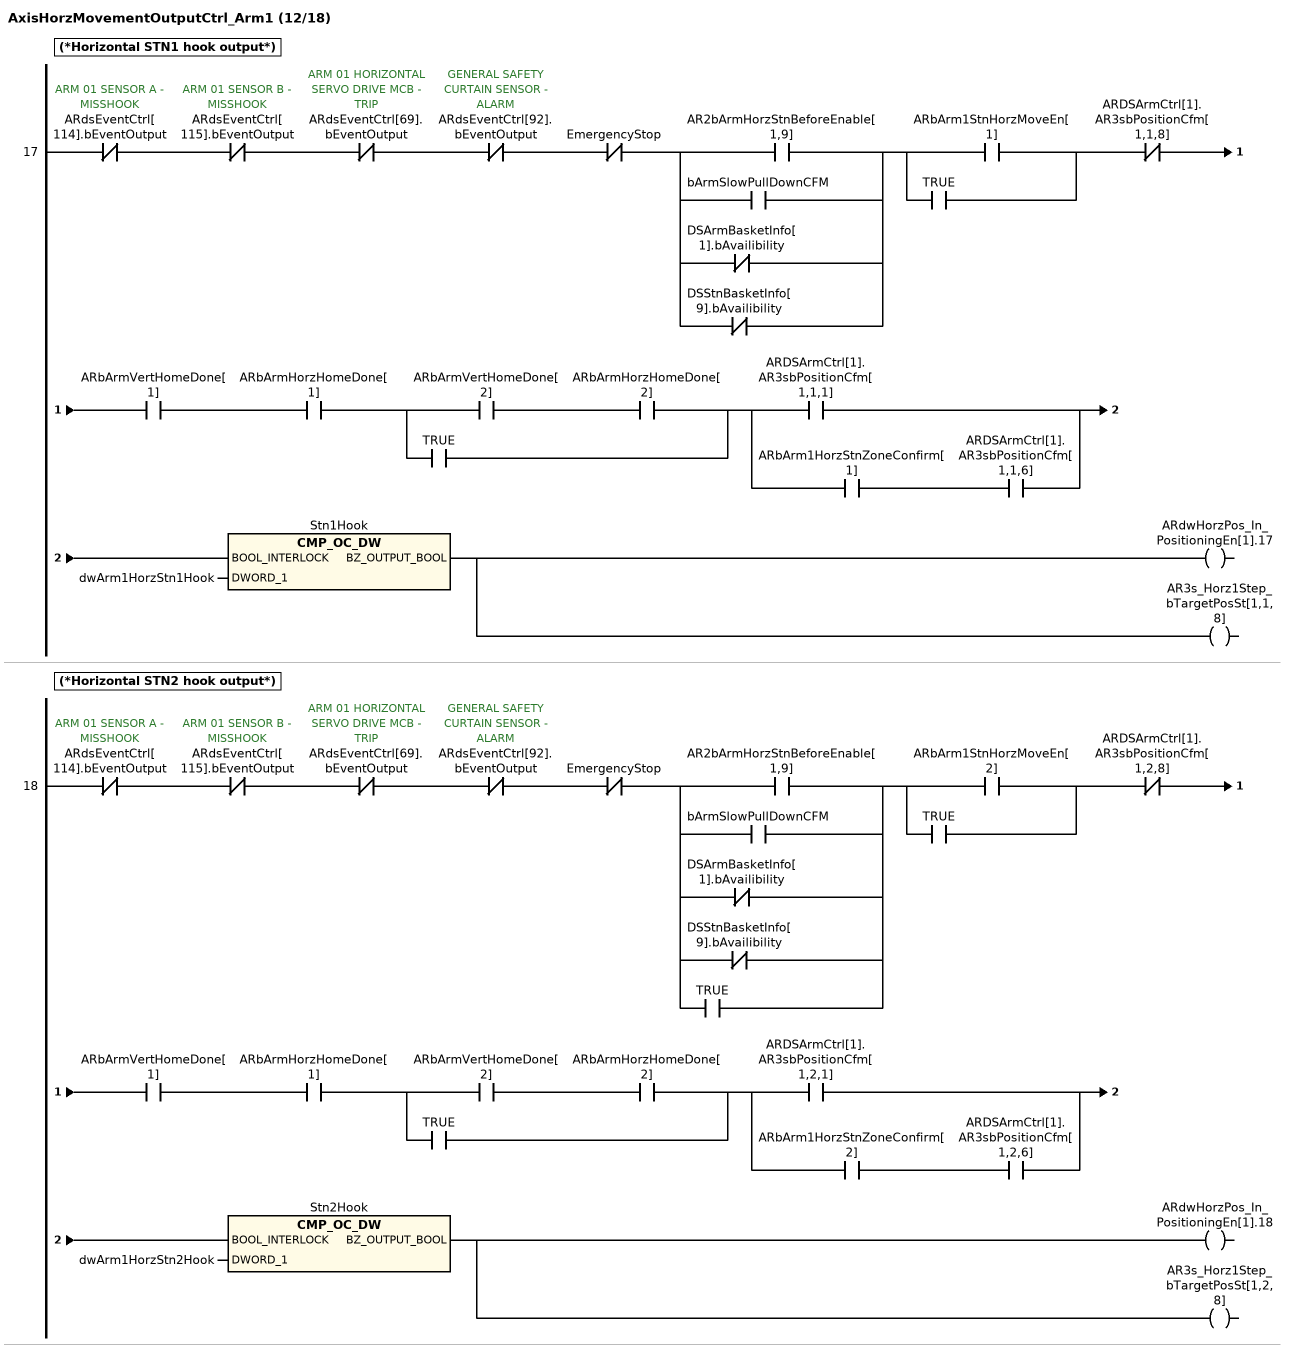
// NETWORK 17
//   ARdsEventCtrl[114].bEventOutput: ARM 01 SENSOR A - MISSHOOK
//   ARdsEventCtrl[115].bEventOutput: ARM 01 SENSOR B - MISSHOOK
//   ARdsEventCtrl[69].bEventOutput: ARM 01 HORIZONTAL SERVO DRIVE MCB - TRIP
//   ARdsEventCtrl[92].bEventOutput: GENERAL SAFETY CURTAIN SENSOR - ALARM
// label: (*Horizontal STN1 hook output*)
Stn1Hook(BOOL_INTERLOCK := ((NOT ARdsEventCtrl[114].bEventOutput AND NOT ARdsEventCtrl[115].bEventOutput AND NOT ARdsEventCtrl[69].bEventOutput AND NOT ARdsEventCtrl[92].bEventOutput AND NOT EmergencyStop) AND (AR2bArmHorzStnBeforeEnable[1,9] OR bArmSlowPullDownCFM OR NOT DSArmBasketInfo[1].bAvailibility OR NOT DSStnBasketInfo[9].bAvailibility) AND (ARbArm1StnHorzMoveEn[1] OR TRUE)) AND NOT ARDSArmCtrl[1].AR3sbPositionCfm[1,1,8] AND ARbArmVertHomeDone[1] AND ARbArmHorzHomeDone[1] AND (ARbArmVertHomeDone[2] AND ARbArmHorzHomeDone[2] OR TRUE) AND (ARDSArmCtrl[1].AR3sbPositionCfm[1,1,1] OR ARbArm1HorzStnZoneConfirm[1] AND ARDSArmCtrl[1].AR3sbPositionCfm[1,1,6]), DWORD_1 := dwArm1HorzStn1Hook); // CMP_OC_DW
ARdwHorzPos_In_PositioningEn[1].17 := Stn1Hook.BZ_OUTPUT_BOOL;
AR3s_Horz1Step_bTargetPosSt[1,1,8] := Stn1Hook.BZ_OUTPUT_BOOL;

// NETWORK 18
//   ARdsEventCtrl[114].bEventOutput: ARM 01 SENSOR A - MISSHOOK
//   ARdsEventCtrl[115].bEventOutput: ARM 01 SENSOR B - MISSHOOK
//   ARdsEventCtrl[69].bEventOutput: ARM 01 HORIZONTAL SERVO DRIVE MCB - TRIP
//   ARdsEventCtrl[92].bEventOutput: GENERAL SAFETY CURTAIN SENSOR - ALARM
// label: (*Horizontal STN2 hook output*)
Stn2Hook(BOOL_INTERLOCK := ((NOT ARdsEventCtrl[114].bEventOutput AND NOT ARdsEventCtrl[115].bEventOutput AND NOT ARdsEventCtrl[69].bEventOutput AND NOT ARdsEventCtrl[92].bEventOutput AND NOT EmergencyStop) AND (AR2bArmHorzStnBeforeEnable[1,9] OR bArmSlowPullDownCFM OR NOT DSArmBasketInfo[1].bAvailibility OR NOT DSStnBasketInfo[9].bAvailibility OR TRUE) AND (ARbArm1StnHorzMoveEn[2] OR TRUE)) AND NOT ARDSArmCtrl[1].AR3sbPositionCfm[1,2,8] AND ARbArmVertHomeDone[1] AND ARbArmHorzHomeDone[1] AND (ARbArmVertHomeDone[2] AND ARbArmHorzHomeDone[2] OR TRUE) AND (ARDSArmCtrl[1].AR3sbPositionCfm[1,2,1] OR ARbArm1HorzStnZoneConfirm[2] AND ARDSArmCtrl[1].AR3sbPositionCfm[1,2,6]), DWORD_1 := dwArm1HorzStn2Hook); // CMP_OC_DW
ARdwHorzPos_In_PositioningEn[1].18 := Stn2Hook.BZ_OUTPUT_BOOL;
AR3s_Horz1Step_bTargetPosSt[1,2,8] := Stn2Hook.BZ_OUTPUT_BOOL;

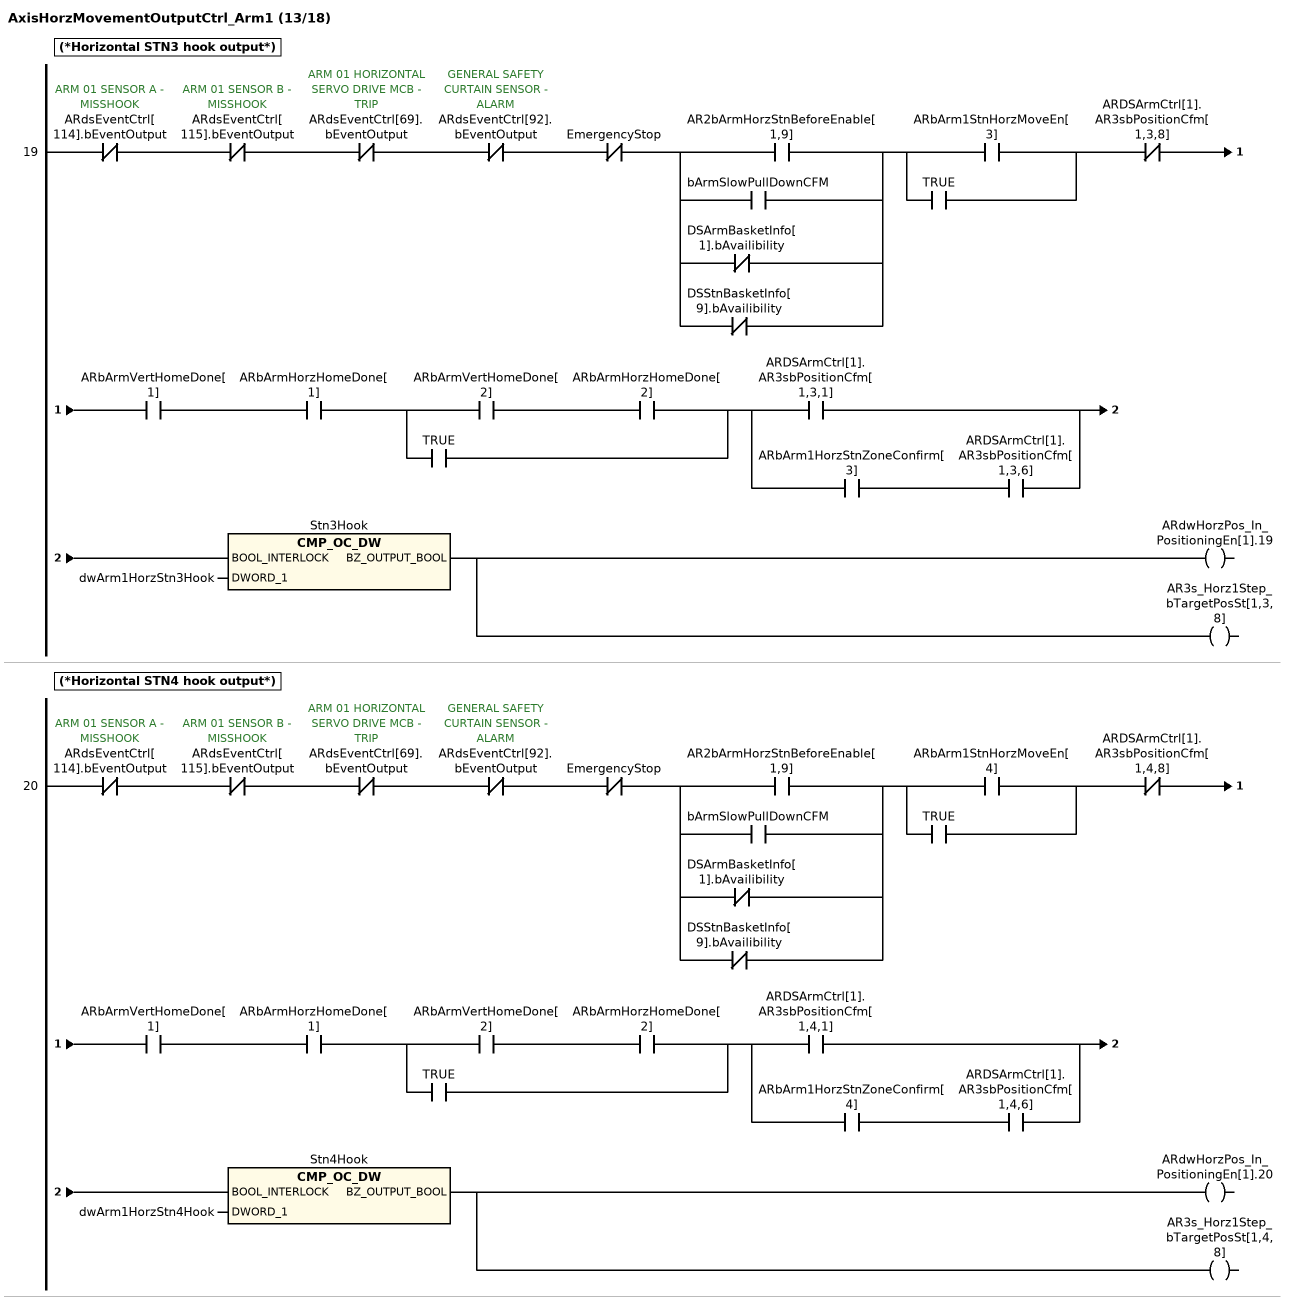
// NETWORK 19
//   ARdsEventCtrl[114].bEventOutput: ARM 01 SENSOR A - MISSHOOK
//   ARdsEventCtrl[115].bEventOutput: ARM 01 SENSOR B - MISSHOOK
//   ARdsEventCtrl[69].bEventOutput: ARM 01 HORIZONTAL SERVO DRIVE MCB - TRIP
//   ARdsEventCtrl[92].bEventOutput: GENERAL SAFETY CURTAIN SENSOR - ALARM
// label: (*Horizontal STN3 hook output*)
Stn3Hook(BOOL_INTERLOCK := ((NOT ARdsEventCtrl[114].bEventOutput AND NOT ARdsEventCtrl[115].bEventOutput AND NOT ARdsEventCtrl[69].bEventOutput AND NOT ARdsEventCtrl[92].bEventOutput AND NOT EmergencyStop) AND (AR2bArmHorzStnBeforeEnable[1,9] OR bArmSlowPullDownCFM OR NOT DSArmBasketInfo[1].bAvailibility OR NOT DSStnBasketInfo[9].bAvailibility) AND (ARbArm1StnHorzMoveEn[3] OR TRUE)) AND NOT ARDSArmCtrl[1].AR3sbPositionCfm[1,3,8] AND ARbArmVertHomeDone[1] AND ARbArmHorzHomeDone[1] AND (ARbArmVertHomeDone[2] AND ARbArmHorzHomeDone[2] OR TRUE) AND (ARDSArmCtrl[1].AR3sbPositionCfm[1,3,1] OR ARbArm1HorzStnZoneConfirm[3] AND ARDSArmCtrl[1].AR3sbPositionCfm[1,3,6]), DWORD_1 := dwArm1HorzStn3Hook); // CMP_OC_DW
ARdwHorzPos_In_PositioningEn[1].19 := Stn3Hook.BZ_OUTPUT_BOOL;
AR3s_Horz1Step_bTargetPosSt[1,3,8] := Stn3Hook.BZ_OUTPUT_BOOL;

// NETWORK 20
//   ARdsEventCtrl[114].bEventOutput: ARM 01 SENSOR A - MISSHOOK
//   ARdsEventCtrl[115].bEventOutput: ARM 01 SENSOR B - MISSHOOK
//   ARdsEventCtrl[69].bEventOutput: ARM 01 HORIZONTAL SERVO DRIVE MCB - TRIP
//   ARdsEventCtrl[92].bEventOutput: GENERAL SAFETY CURTAIN SENSOR - ALARM
// label: (*Horizontal STN4 hook output*)
Stn4Hook(BOOL_INTERLOCK := ((NOT ARdsEventCtrl[114].bEventOutput AND NOT ARdsEventCtrl[115].bEventOutput AND NOT ARdsEventCtrl[69].bEventOutput AND NOT ARdsEventCtrl[92].bEventOutput AND NOT EmergencyStop) AND (AR2bArmHorzStnBeforeEnable[1,9] OR bArmSlowPullDownCFM OR NOT DSArmBasketInfo[1].bAvailibility OR NOT DSStnBasketInfo[9].bAvailibility) AND (ARbArm1StnHorzMoveEn[4] OR TRUE)) AND NOT ARDSArmCtrl[1].AR3sbPositionCfm[1,4,8] AND ARbArmVertHomeDone[1] AND ARbArmHorzHomeDone[1] AND (ARbArmVertHomeDone[2] AND ARbArmHorzHomeDone[2] OR TRUE) AND (ARDSArmCtrl[1].AR3sbPositionCfm[1,4,1] OR ARbArm1HorzStnZoneConfirm[4] AND ARDSArmCtrl[1].AR3sbPositionCfm[1,4,6]), DWORD_1 := dwArm1HorzStn4Hook); // CMP_OC_DW
ARdwHorzPos_In_PositioningEn[1].20 := Stn4Hook.BZ_OUTPUT_BOOL;
AR3s_Horz1Step_bTargetPosSt[1,4,8] := Stn4Hook.BZ_OUTPUT_BOOL;

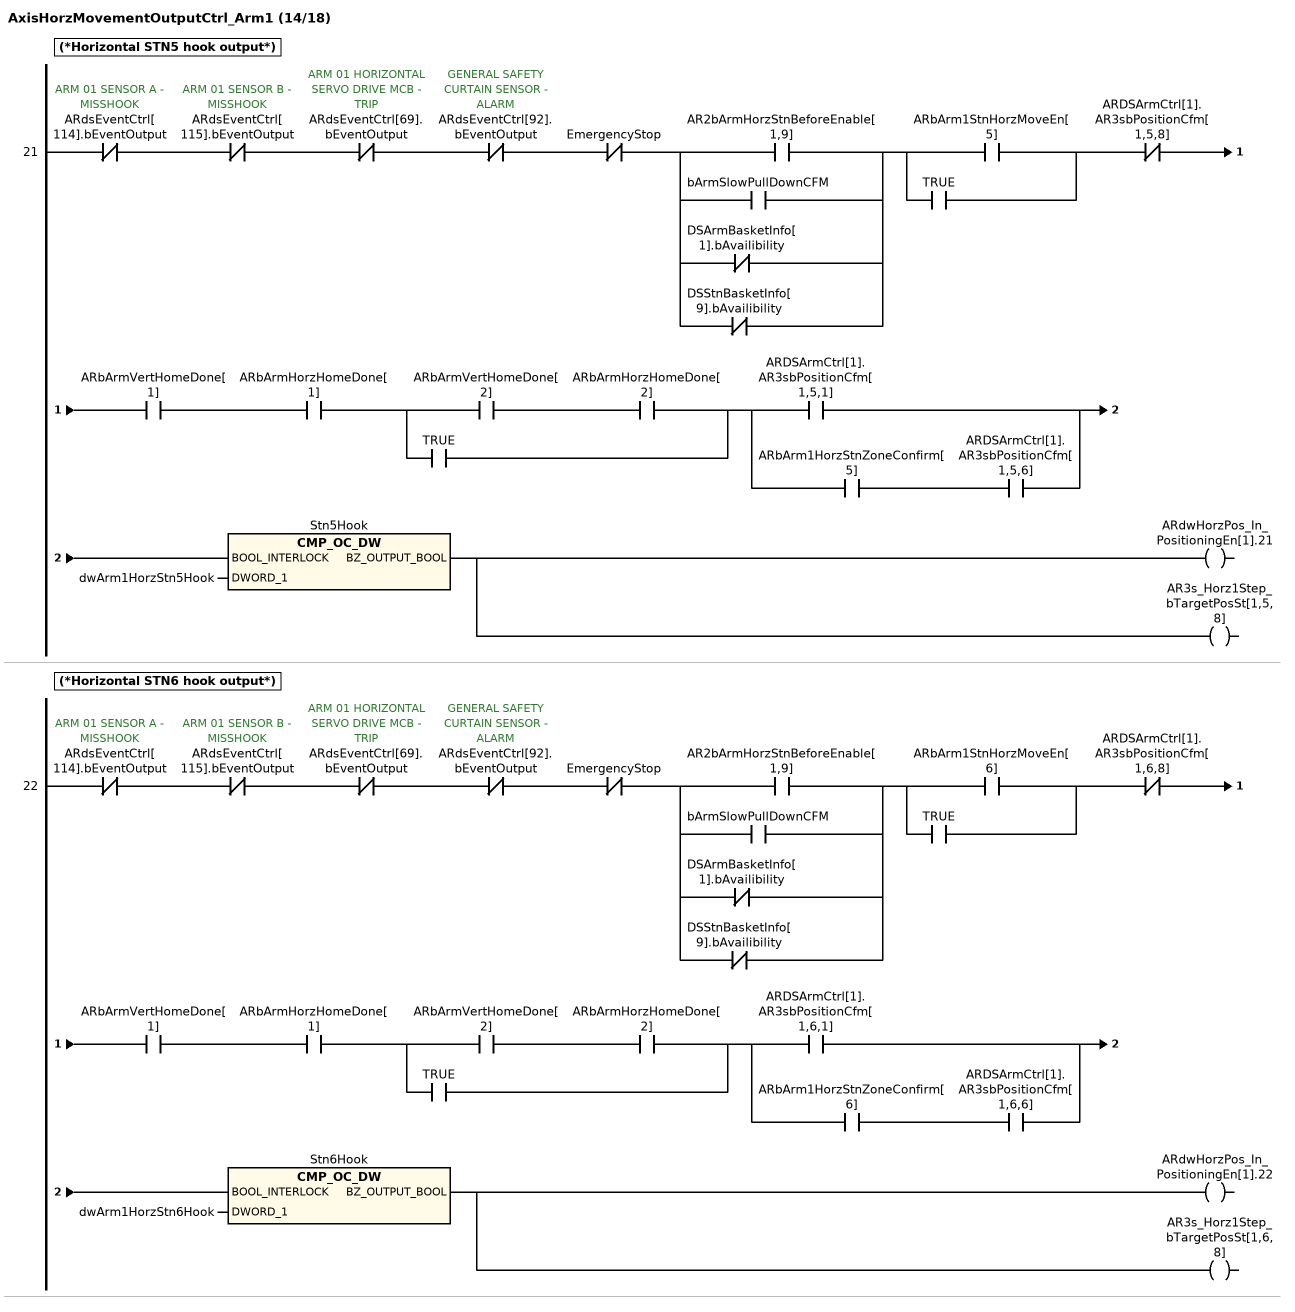
// NETWORK 21
//   ARdsEventCtrl[114].bEventOutput: ARM 01 SENSOR A - MISSHOOK
//   ARdsEventCtrl[115].bEventOutput: ARM 01 SENSOR B - MISSHOOK
//   ARdsEventCtrl[69].bEventOutput: ARM 01 HORIZONTAL SERVO DRIVE MCB - TRIP
//   ARdsEventCtrl[92].bEventOutput: GENERAL SAFETY CURTAIN SENSOR - ALARM
// label: (*Horizontal STN5 hook output*)
Stn5Hook(BOOL_INTERLOCK := ((NOT ARdsEventCtrl[114].bEventOutput AND NOT ARdsEventCtrl[115].bEventOutput AND NOT ARdsEventCtrl[69].bEventOutput AND NOT ARdsEventCtrl[92].bEventOutput AND NOT EmergencyStop) AND (AR2bArmHorzStnBeforeEnable[1,9] OR bArmSlowPullDownCFM OR NOT DSArmBasketInfo[1].bAvailibility OR NOT DSStnBasketInfo[9].bAvailibility) AND (ARbArm1StnHorzMoveEn[5] OR TRUE)) AND NOT ARDSArmCtrl[1].AR3sbPositionCfm[1,5,8] AND ARbArmVertHomeDone[1] AND ARbArmHorzHomeDone[1] AND (ARbArmVertHomeDone[2] AND ARbArmHorzHomeDone[2] OR TRUE) AND (ARDSArmCtrl[1].AR3sbPositionCfm[1,5,1] OR ARbArm1HorzStnZoneConfirm[5] AND ARDSArmCtrl[1].AR3sbPositionCfm[1,5,6]), DWORD_1 := dwArm1HorzStn5Hook); // CMP_OC_DW
ARdwHorzPos_In_PositioningEn[1].21 := Stn5Hook.BZ_OUTPUT_BOOL;
AR3s_Horz1Step_bTargetPosSt[1,5,8] := Stn5Hook.BZ_OUTPUT_BOOL;

// NETWORK 22
//   ARdsEventCtrl[114].bEventOutput: ARM 01 SENSOR A - MISSHOOK
//   ARdsEventCtrl[115].bEventOutput: ARM 01 SENSOR B - MISSHOOK
//   ARdsEventCtrl[69].bEventOutput: ARM 01 HORIZONTAL SERVO DRIVE MCB - TRIP
//   ARdsEventCtrl[92].bEventOutput: GENERAL SAFETY CURTAIN SENSOR - ALARM
// label: (*Horizontal STN6 hook output*)
Stn6Hook(BOOL_INTERLOCK := ((NOT ARdsEventCtrl[114].bEventOutput AND NOT ARdsEventCtrl[115].bEventOutput AND NOT ARdsEventCtrl[69].bEventOutput AND NOT ARdsEventCtrl[92].bEventOutput AND NOT EmergencyStop) AND ((AR2bArmHorzStnBeforeEnable[1,9] OR bArmSlowPullDownCFM OR NOT DSArmBasketInfo[1].bAvailibility OR NOT DSStnBasketInfo[9].bAvailibility) AND (ARbArm1StnHorzMoveEn[6] OR TRUE))) AND NOT ARDSArmCtrl[1].AR3sbPositionCfm[1,6,8] AND ARbArmVertHomeDone[1] AND ARbArmHorzHomeDone[1] AND (ARbArmVertHomeDone[2] AND ARbArmHorzHomeDone[2] OR TRUE) AND (ARDSArmCtrl[1].AR3sbPositionCfm[1,6,1] OR ARbArm1HorzStnZoneConfirm[6] AND ARDSArmCtrl[1].AR3sbPositionCfm[1,6,6]), DWORD_1 := dwArm1HorzStn6Hook); // CMP_OC_DW
ARdwHorzPos_In_PositioningEn[1].22 := Stn6Hook.BZ_OUTPUT_BOOL;
AR3s_Horz1Step_bTargetPosSt[1,6,8] := Stn6Hook.BZ_OUTPUT_BOOL;

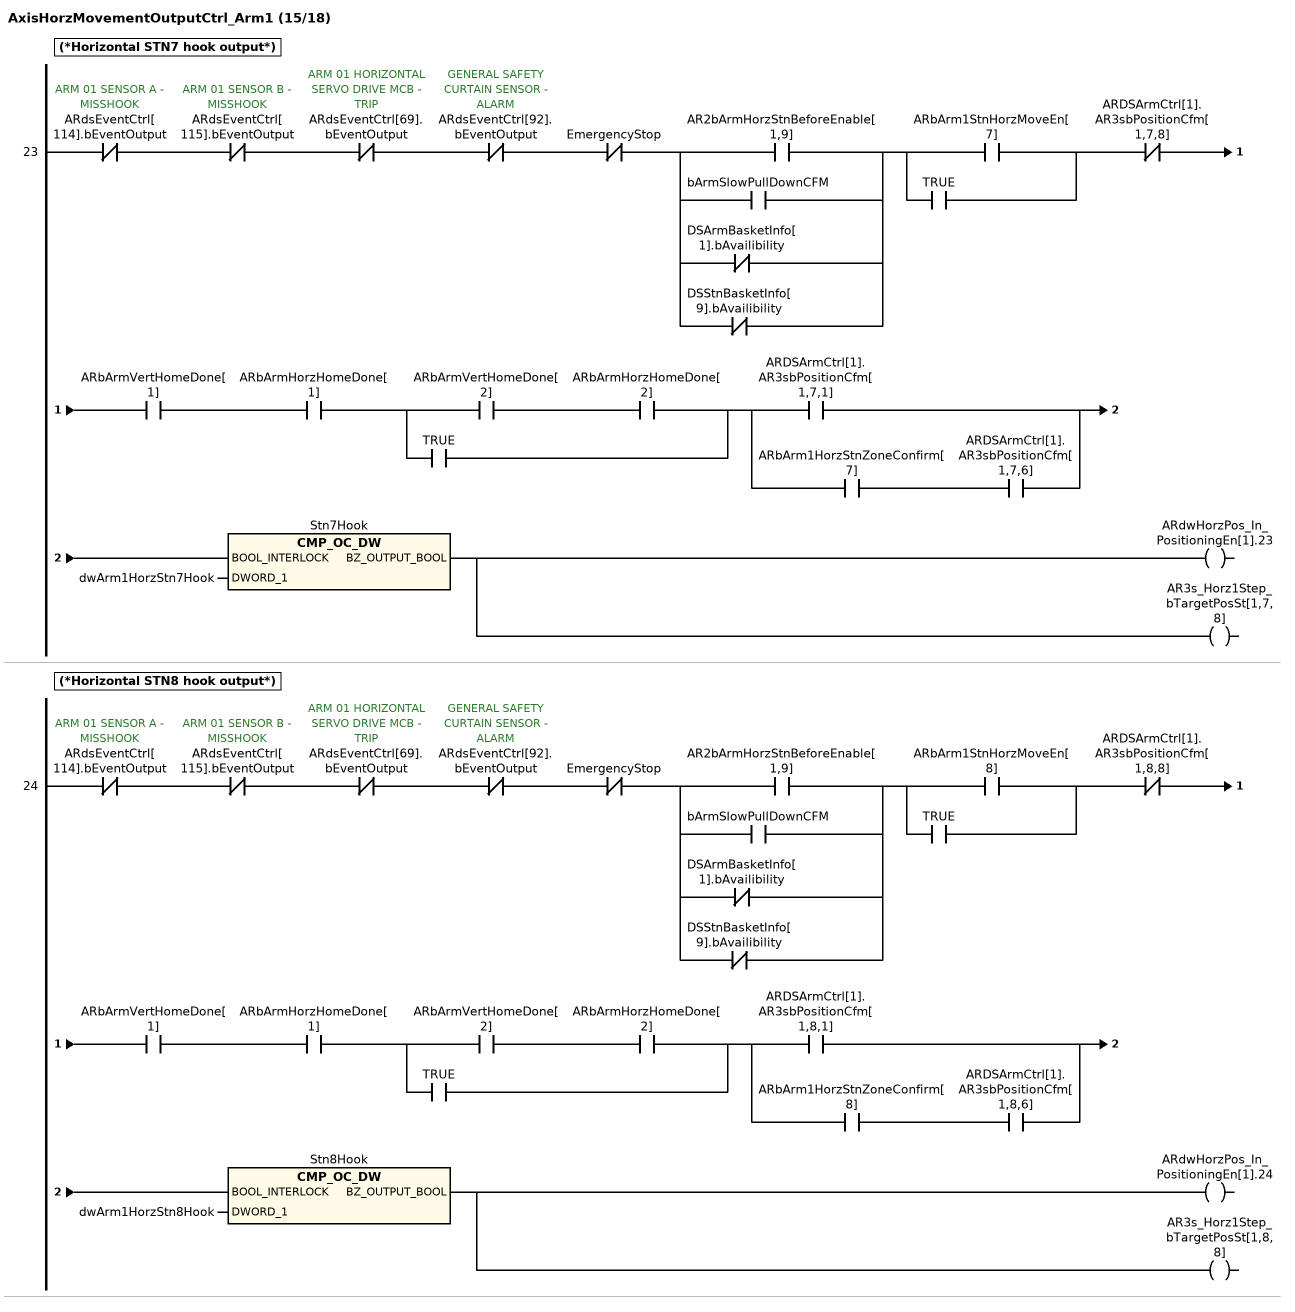
// NETWORK 23
//   ARdsEventCtrl[114].bEventOutput: ARM 01 SENSOR A - MISSHOOK
//   ARdsEventCtrl[115].bEventOutput: ARM 01 SENSOR B - MISSHOOK
//   ARdsEventCtrl[69].bEventOutput: ARM 01 HORIZONTAL SERVO DRIVE MCB - TRIP
//   ARdsEventCtrl[92].bEventOutput: GENERAL SAFETY CURTAIN SENSOR - ALARM
// label: (*Horizontal STN7 hook output*)
Stn7Hook(BOOL_INTERLOCK := ((NOT ARdsEventCtrl[114].bEventOutput AND NOT ARdsEventCtrl[115].bEventOutput AND NOT ARdsEventCtrl[69].bEventOutput AND NOT ARdsEventCtrl[92].bEventOutput AND NOT EmergencyStop) AND (AR2bArmHorzStnBeforeEnable[1,9] OR bArmSlowPullDownCFM OR NOT DSArmBasketInfo[1].bAvailibility OR NOT DSStnBasketInfo[9].bAvailibility) AND (ARbArm1StnHorzMoveEn[7] OR TRUE)) AND NOT ARDSArmCtrl[1].AR3sbPositionCfm[1,7,8] AND ARbArmVertHomeDone[1] AND ARbArmHorzHomeDone[1] AND (ARbArmVertHomeDone[2] AND ARbArmHorzHomeDone[2] OR TRUE) AND (ARDSArmCtrl[1].AR3sbPositionCfm[1,7,1] OR ARbArm1HorzStnZoneConfirm[7] AND ARDSArmCtrl[1].AR3sbPositionCfm[1,7,6]), DWORD_1 := dwArm1HorzStn7Hook); // CMP_OC_DW
ARdwHorzPos_In_PositioningEn[1].23 := Stn7Hook.BZ_OUTPUT_BOOL;
AR3s_Horz1Step_bTargetPosSt[1,7,8] := Stn7Hook.BZ_OUTPUT_BOOL;

// NETWORK 24
//   ARdsEventCtrl[114].bEventOutput: ARM 01 SENSOR A - MISSHOOK
//   ARdsEventCtrl[115].bEventOutput: ARM 01 SENSOR B - MISSHOOK
//   ARdsEventCtrl[69].bEventOutput: ARM 01 HORIZONTAL SERVO DRIVE MCB - TRIP
//   ARdsEventCtrl[92].bEventOutput: GENERAL SAFETY CURTAIN SENSOR - ALARM
// label: (*Horizontal STN8 hook output*)
Stn8Hook(BOOL_INTERLOCK := (NOT ARdsEventCtrl[114].bEventOutput AND NOT ARdsEventCtrl[115].bEventOutput AND NOT ARdsEventCtrl[69].bEventOutput AND NOT ARdsEventCtrl[92].bEventOutput AND NOT EmergencyStop AND (AR2bArmHorzStnBeforeEnable[1,9] OR bArmSlowPullDownCFM OR NOT DSArmBasketInfo[1].bAvailibility OR NOT DSStnBasketInfo[9].bAvailibility) AND (ARbArm1StnHorzMoveEn[8] OR TRUE)) AND NOT ARDSArmCtrl[1].AR3sbPositionCfm[1,8,8] AND ARbArmVertHomeDone[1] AND ARbArmHorzHomeDone[1] AND (ARbArmVertHomeDone[2] AND ARbArmHorzHomeDone[2] OR TRUE) AND (ARDSArmCtrl[1].AR3sbPositionCfm[1,8,1] OR ARbArm1HorzStnZoneConfirm[8] AND ARDSArmCtrl[1].AR3sbPositionCfm[1,8,6]), DWORD_1 := dwArm1HorzStn8Hook); // CMP_OC_DW
ARdwHorzPos_In_PositioningEn[1].24 := Stn8Hook.BZ_OUTPUT_BOOL;
AR3s_Horz1Step_bTargetPosSt[1,8,8] := Stn8Hook.BZ_OUTPUT_BOOL;

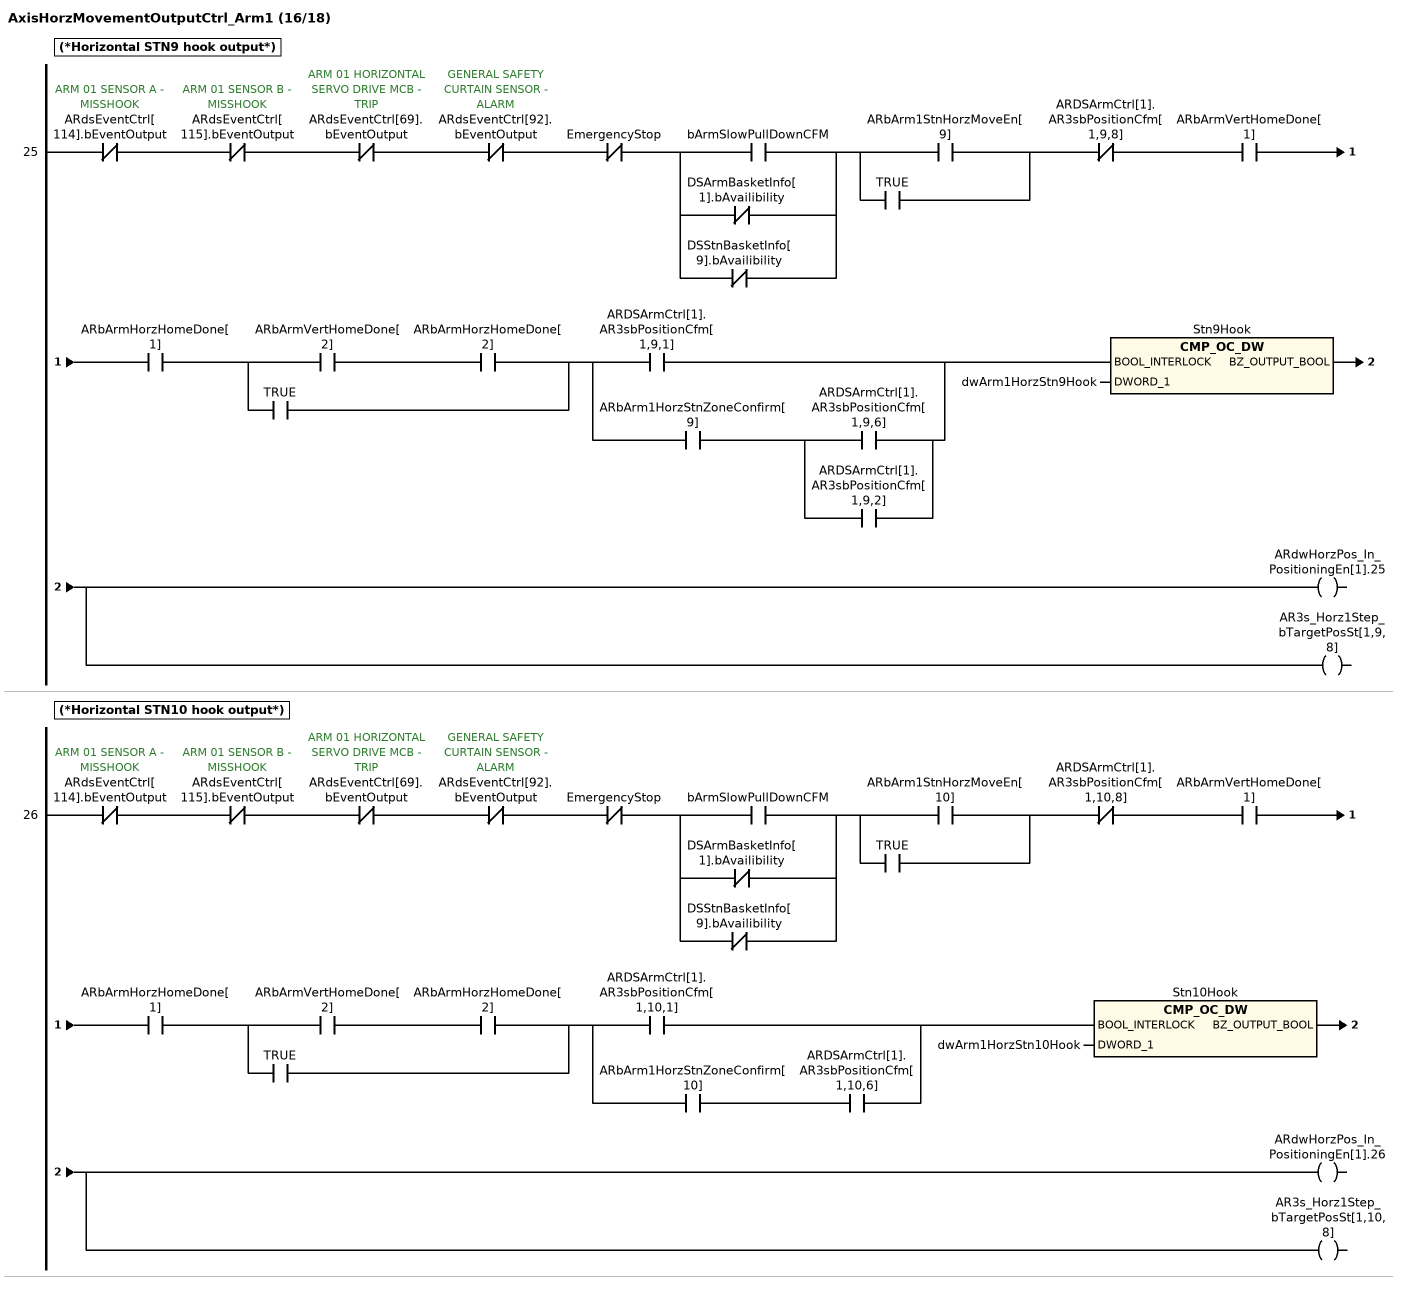
// NETWORK 25
//   ARdsEventCtrl[114].bEventOutput: ARM 01 SENSOR A - MISSHOOK
//   ARdsEventCtrl[115].bEventOutput: ARM 01 SENSOR B - MISSHOOK
//   ARdsEventCtrl[69].bEventOutput: ARM 01 HORIZONTAL SERVO DRIVE MCB - TRIP
//   ARdsEventCtrl[92].bEventOutput: GENERAL SAFETY CURTAIN SENSOR - ALARM
// label: (*Horizontal STN9 hook output*)
Stn9Hook(BOOL_INTERLOCK := ((NOT ARdsEventCtrl[114].bEventOutput AND NOT ARdsEventCtrl[115].bEventOutput AND NOT ARdsEventCtrl[69].bEventOutput AND NOT ARdsEventCtrl[92].bEventOutput AND NOT EmergencyStop) AND (bArmSlowPullDownCFM OR NOT DSArmBasketInfo[1].bAvailibility OR NOT DSStnBasketInfo[9].bAvailibility) AND (ARbArm1StnHorzMoveEn[9] OR TRUE)) AND NOT ARDSArmCtrl[1].AR3sbPositionCfm[1,9,8] AND ARbArmVertHomeDone[1] AND ARbArmHorzHomeDone[1] AND (ARbArmVertHomeDone[2] AND ARbArmHorzHomeDone[2] OR TRUE) AND (ARDSArmCtrl[1].AR3sbPositionCfm[1,9,1] OR ARbArm1HorzStnZoneConfirm[9] AND (ARDSArmCtrl[1].AR3sbPositionCfm[1,9,6] OR ARDSArmCtrl[1].AR3sbPositionCfm[1,9,2])), DWORD_1 := dwArm1HorzStn9Hook); // CMP_OC_DW
ARdwHorzPos_In_PositioningEn[1].25 := Stn9Hook.BZ_OUTPUT_BOOL;
AR3s_Horz1Step_bTargetPosSt[1,9,8] := Stn9Hook.BZ_OUTPUT_BOOL;

// NETWORK 26
//   ARdsEventCtrl[114].bEventOutput: ARM 01 SENSOR A - MISSHOOK
//   ARdsEventCtrl[115].bEventOutput: ARM 01 SENSOR B - MISSHOOK
//   ARdsEventCtrl[69].bEventOutput: ARM 01 HORIZONTAL SERVO DRIVE MCB - TRIP
//   ARdsEventCtrl[92].bEventOutput: GENERAL SAFETY CURTAIN SENSOR - ALARM
// label: (*Horizontal STN10 hook output*)
Stn10Hook(BOOL_INTERLOCK := ((NOT ARdsEventCtrl[114].bEventOutput AND NOT ARdsEventCtrl[115].bEventOutput AND NOT ARdsEventCtrl[69].bEventOutput AND NOT ARdsEventCtrl[92].bEventOutput AND NOT EmergencyStop) AND (bArmSlowPullDownCFM OR NOT DSArmBasketInfo[1].bAvailibility OR NOT DSStnBasketInfo[9].bAvailibility) AND (ARbArm1StnHorzMoveEn[10] OR TRUE)) AND NOT ARDSArmCtrl[1].AR3sbPositionCfm[1,10,8] AND ARbArmVertHomeDone[1] AND ARbArmHorzHomeDone[1] AND (ARbArmVertHomeDone[2] AND ARbArmHorzHomeDone[2] OR TRUE) AND (ARDSArmCtrl[1].AR3sbPositionCfm[1,10,1] OR ARbArm1HorzStnZoneConfirm[10] AND ARDSArmCtrl[1].AR3sbPositionCfm[1,10,6]), DWORD_1 := dwArm1HorzStn10Hook); // CMP_OC_DW
ARdwHorzPos_In_PositioningEn[1].26 := Stn10Hook.BZ_OUTPUT_BOOL;
AR3s_Horz1Step_bTargetPosSt[1,10,8] := Stn10Hook.BZ_OUTPUT_BOOL;

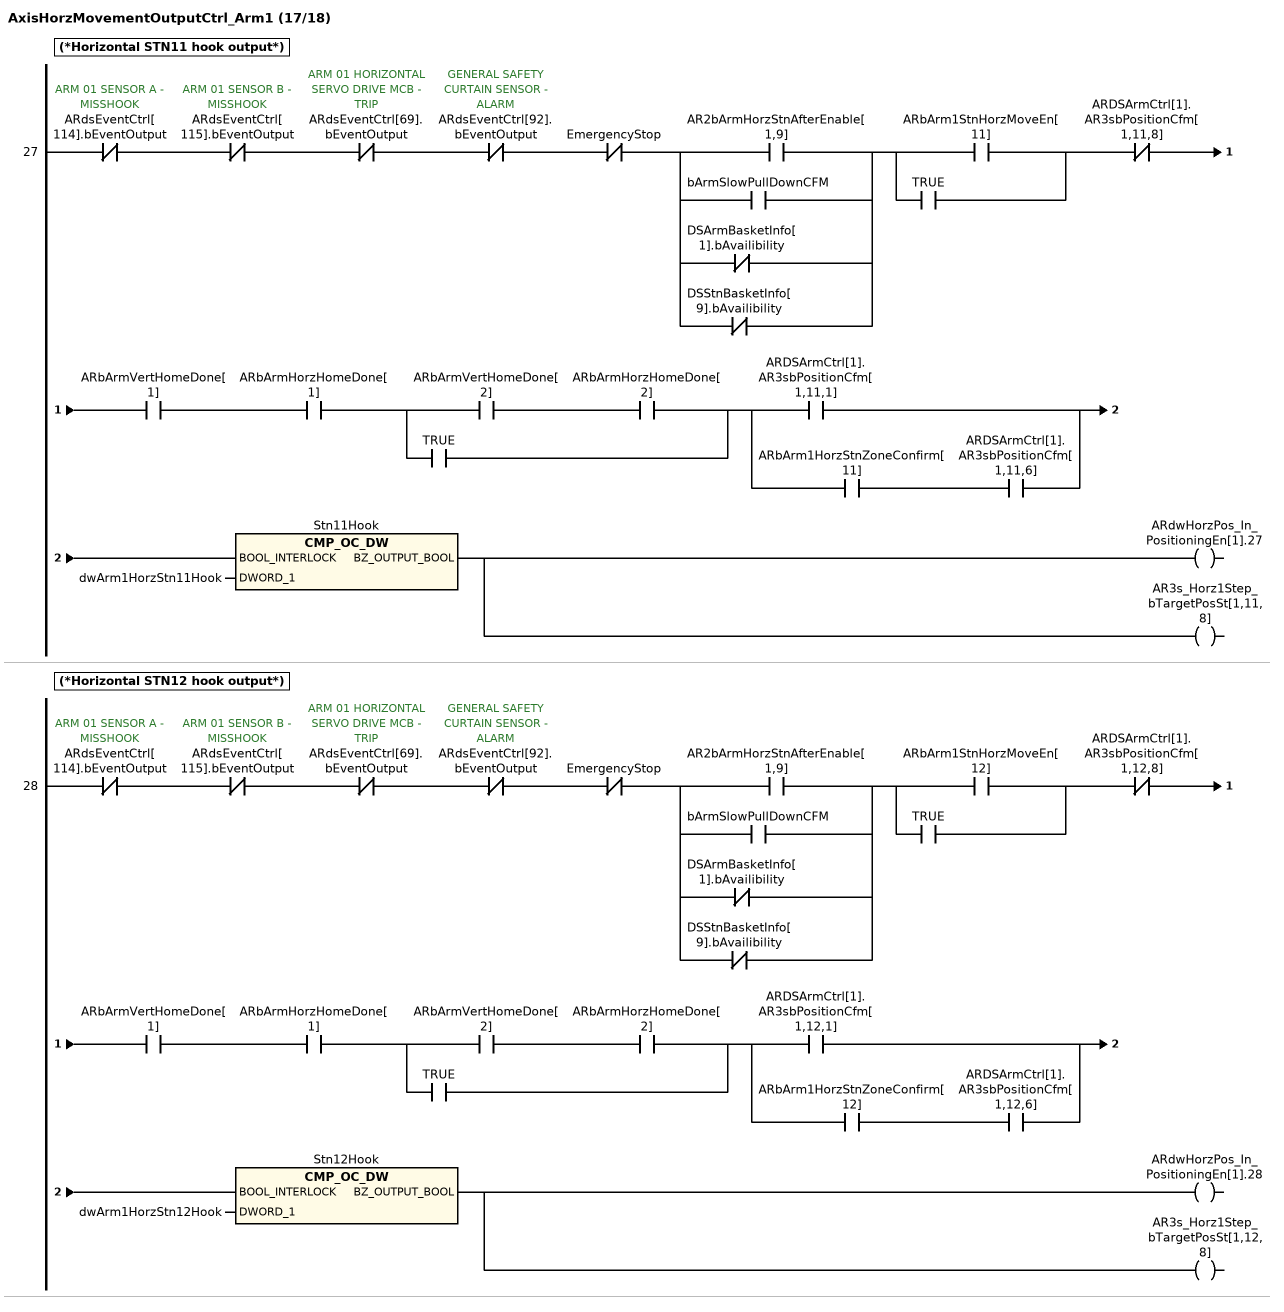
// NETWORK 27
//   ARdsEventCtrl[114].bEventOutput: ARM 01 SENSOR A - MISSHOOK
//   ARdsEventCtrl[115].bEventOutput: ARM 01 SENSOR B - MISSHOOK
//   ARdsEventCtrl[69].bEventOutput: ARM 01 HORIZONTAL SERVO DRIVE MCB - TRIP
//   ARdsEventCtrl[92].bEventOutput: GENERAL SAFETY CURTAIN SENSOR - ALARM
// label: (*Horizontal STN11 hook output*)
Stn11Hook(BOOL_INTERLOCK := ((NOT ARdsEventCtrl[114].bEventOutput AND NOT ARdsEventCtrl[115].bEventOutput AND NOT ARdsEventCtrl[69].bEventOutput AND NOT ARdsEventCtrl[92].bEventOutput AND NOT EmergencyStop) AND (AR2bArmHorzStnAfterEnable[1,9] OR bArmSlowPullDownCFM OR NOT DSArmBasketInfo[1].bAvailibility OR NOT DSStnBasketInfo[9].bAvailibility) AND (ARbArm1StnHorzMoveEn[11] OR TRUE)) AND NOT ARDSArmCtrl[1].AR3sbPositionCfm[1,11,8] AND ARbArmVertHomeDone[1] AND ARbArmHorzHomeDone[1] AND (ARbArmVertHomeDone[2] AND ARbArmHorzHomeDone[2] OR TRUE) AND (ARDSArmCtrl[1].AR3sbPositionCfm[1,11,1] OR ARbArm1HorzStnZoneConfirm[11] AND ARDSArmCtrl[1].AR3sbPositionCfm[1,11,6]), DWORD_1 := dwArm1HorzStn11Hook); // CMP_OC_DW
ARdwHorzPos_In_PositioningEn[1].27 := Stn11Hook.BZ_OUTPUT_BOOL;
AR3s_Horz1Step_bTargetPosSt[1,11,8] := Stn11Hook.BZ_OUTPUT_BOOL;

// NETWORK 28
//   ARdsEventCtrl[114].bEventOutput: ARM 01 SENSOR A - MISSHOOK
//   ARdsEventCtrl[115].bEventOutput: ARM 01 SENSOR B - MISSHOOK
//   ARdsEventCtrl[69].bEventOutput: ARM 01 HORIZONTAL SERVO DRIVE MCB - TRIP
//   ARdsEventCtrl[92].bEventOutput: GENERAL SAFETY CURTAIN SENSOR - ALARM
// label: (*Horizontal STN12 hook output*)
Stn12Hook(BOOL_INTERLOCK := ((NOT ARdsEventCtrl[114].bEventOutput AND NOT ARdsEventCtrl[115].bEventOutput AND NOT ARdsEventCtrl[69].bEventOutput AND NOT ARdsEventCtrl[92].bEventOutput AND NOT EmergencyStop) AND (AR2bArmHorzStnAfterEnable[1,9] OR bArmSlowPullDownCFM OR NOT DSArmBasketInfo[1].bAvailibility OR NOT DSStnBasketInfo[9].bAvailibility) AND (ARbArm1StnHorzMoveEn[12] OR TRUE)) AND NOT ARDSArmCtrl[1].AR3sbPositionCfm[1,12,8] AND ARbArmVertHomeDone[1] AND ARbArmHorzHomeDone[1] AND (ARbArmVertHomeDone[2] AND ARbArmHorzHomeDone[2] OR TRUE) AND (ARDSArmCtrl[1].AR3sbPositionCfm[1,12,1] OR ARbArm1HorzStnZoneConfirm[12] AND ARDSArmCtrl[1].AR3sbPositionCfm[1,12,6]), DWORD_1 := dwArm1HorzStn12Hook); // CMP_OC_DW
ARdwHorzPos_In_PositioningEn[1].28 := Stn12Hook.BZ_OUTPUT_BOOL;
AR3s_Horz1Step_bTargetPosSt[1,12,8] := Stn12Hook.BZ_OUTPUT_BOOL;

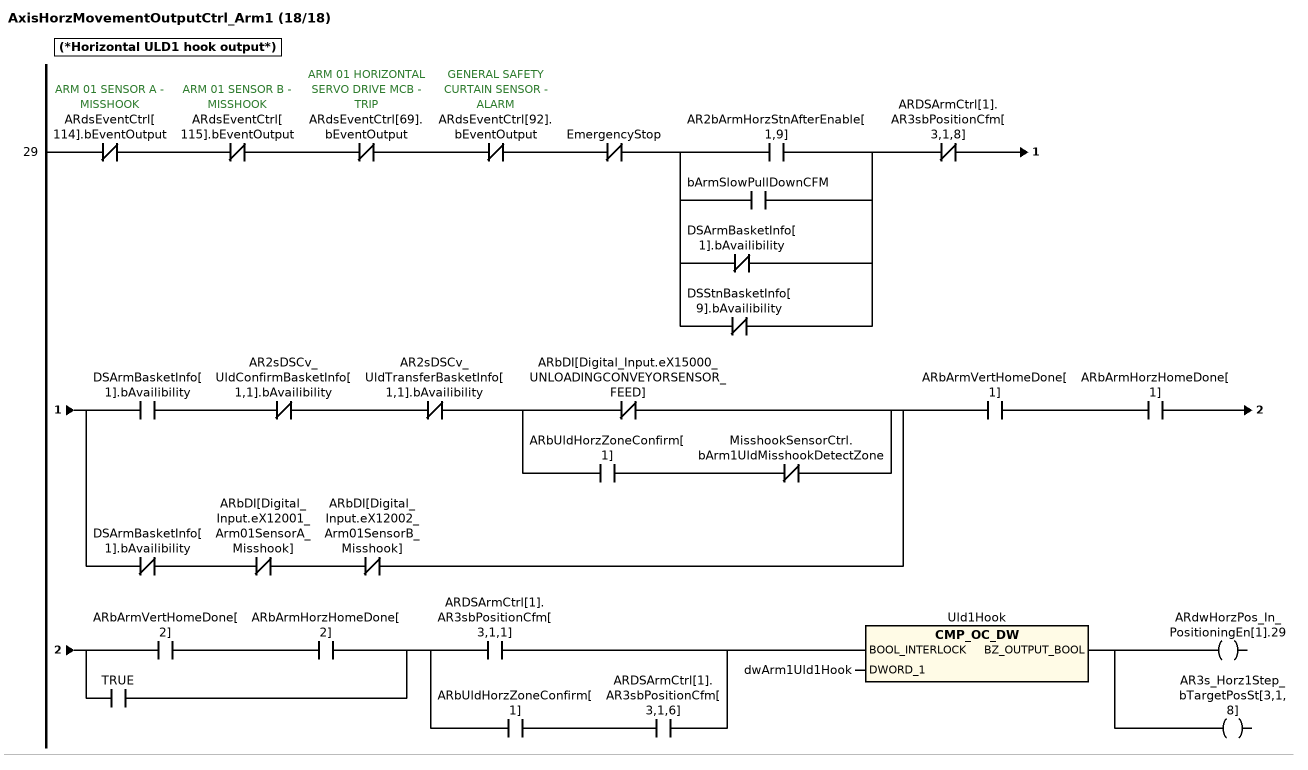
// NETWORK 29
//   ARdsEventCtrl[114].bEventOutput: ARM 01 SENSOR A - MISSHOOK
//   ARdsEventCtrl[115].bEventOutput: ARM 01 SENSOR B - MISSHOOK
//   ARdsEventCtrl[69].bEventOutput: ARM 01 HORIZONTAL SERVO DRIVE MCB - TRIP
//   ARdsEventCtrl[92].bEventOutput: GENERAL SAFETY CURTAIN SENSOR - ALARM
// label: (*Horizontal ULD1 hook output*)
Uld1Hook(BOOL_INTERLOCK := (((NOT ARdsEventCtrl[114].bEventOutput AND NOT ARdsEventCtrl[115].bEventOutput AND NOT ARdsEventCtrl[69].bEventOutput AND NOT ARdsEventCtrl[92].bEventOutput AND NOT EmergencyStop) AND (AR2bArmHorzStnAfterEnable[1,9] OR bArmSlowPullDownCFM OR NOT DSArmBasketInfo[1].bAvailibility OR NOT DSStnBasketInfo[9].bAvailibility)) AND NOT ARDSArmCtrl[1].AR3sbPositionCfm[3,1,8] AND (DSArmBasketInfo[1].bAvailibility AND NOT AR2sDSCv_UldConfirmBasketInfo[1,1].bAvailibility AND NOT AR2sDSCv_UldTransferBasketInfo[1,1].bAvailibility AND (NOT ARbDI[Digital_Input.eX15000_UNLOADINGCONVEYORSENSOR_FEED] OR ARbUldHorzZoneConfirm[1] AND NOT MisshookSensorCtrl.bArm1UldMisshookDetectZone) OR NOT DSArmBasketInfo[1].bAvailibility AND NOT ARbDI[Digital_Input.eX12001_Arm01SensorA_Misshook] AND NOT ARbDI[Digital_Input.eX12002_Arm01SensorB_Misshook])) AND ARbArmVertHomeDone[1] AND ARbArmHorzHomeDone[1] AND (ARbArmVertHomeDone[2] AND ARbArmHorzHomeDone[2] OR TRUE) AND (ARDSArmCtrl[1].AR3sbPositionCfm[3,1,1] OR ARbUldHorzZoneConfirm[1] AND ARDSArmCtrl[1].AR3sbPositionCfm[3,1,6]), DWORD_1 := dwArm1Uld1Hook); // CMP_OC_DW
ARdwHorzPos_In_PositioningEn[1].29 := Uld1Hook.BZ_OUTPUT_BOOL;
AR3s_Horz1Step_bTargetPosSt[3,1,8] := Uld1Hook.BZ_OUTPUT_BOOL;

END_PROGRAM

(* stored: Version 1.1.0.1, ProductVersion 3.1.4024.12
   POU AxisHorzMovementOutputCtrl_Arm1: Id {70224aff-b3cf-4529-86a3-051e51a6840c}, SpecialFunc None *)
